(* Logix 5000 project; controller reports 1756-L63 rev 20.11; software revision 20.04; part 28 of 52 *)

        [2013].time.Year := 2023, [2013].time.Month := 1, [2013].time.Day := 16, [2013].time.Hour := 16, [2013].time.Minute := 9, [2013].time.Second := 59, [2014].log_data[0].min := 1.0, [2014].log_data[0].max := 1.0, [2014].log_data[0].total := 300.0, [2014].log_data[0].time := 300.0, [2014].log_data[0].minminute := 10, [2014].log_data[0].maxminute := 10, [2014].log_data[0].valid := 1, [2014].log_data[1].valid := 1, [2014].log_data[2].valid := 1, [2014].log_data[3].valid := 1, [2014].log_data[4].valid := 1, [2014].log_data[5].valid := 1, [2014].log_data[6].valid := 1, [2014].log_data[7].valid := 1, [2014].log_data[8].valid := 1, [2014].log_data[9].valid := 1, [2014].log_data[10].valid := 1, [2014].log_data[11].valid := 1, [2014].log_data[12].valid := 1, [2014].log_data[13].valid := 1, [2014].log_data[14].valid := 1, [2014].log_data[15].valid := 1, [2014].log_data[16].valid := 1, [2014].log_data[17].valid := 1, [2014].log_data[18].valid := 1, [2014].log_data[19].valid := 1, [2014].time.Year := 2023, [2014].time.Month := 1, [2014].time.Day := 16, [2014].time.Hour := 16, [2014].time.Minute := 14, [2014].time.Second := 59, [2015].log_data[0].min := 1.0, [2015].log_data[0].max := 1.0, [2015].log_data[0].total := 300.0, [2015].log_data[0].time := 300.0, [2015].log_data[0].minminute := 15, [2015].log_data[0].maxminute := 15, [2015].log_data[0].valid := 1, [2015].log_data[1].valid := 1, [2015].log_data[2].valid := 1, [2015].log_data[3].valid := 1, [2015].log_data[4].valid := 1, [2015].log_data[5].valid := 1, [2015].log_data[6].valid := 1, [2015].log_data[7].valid := 1, [2015].log_data[8].valid := 1, [2015].log_data[9].valid := 1, [2015].log_data[10].valid := 1, [2015].log_data[11].valid := 1, [2015].log_data[12].valid := 1, [2015].log_data[13].valid := 1, [2015].log_data[14].valid := 1, [2015].log_data[15].valid := 1,
        [2015].log_data[16].valid := 1, [2015].log_data[17].valid := 1, [2015].log_data[18].valid := 1, [2015].log_data[19].valid := 1, [2015].time.Year := 2023, [2015].time.Month := 1, [2015].time.Day := 16, [2015].time.Hour := 16, [2015].time.Minute := 19, [2015].time.Second := 59, [2016].log_data[0].min := 1.0, [2016].log_data[0].max := 1.0, [2016].log_data[0].total := 300.0, [2016].log_data[0].time := 300.0, [2016].log_data[0].minminute := 20, [2016].log_data[0].maxminute := 20, [2016].log_data[0].valid := 1, [2016].log_data[1].valid := 1, [2016].log_data[2].valid := 1, [2016].log_data[3].valid := 1, [2016].log_data[4].valid := 1, [2016].log_data[5].valid := 1, [2016].log_data[6].valid := 1, [2016].log_data[7].valid := 1, [2016].log_data[8].valid := 1, [2016].log_data[9].valid := 1, [2016].log_data[10].valid := 1, [2016].log_data[11].valid := 1, [2016].log_data[12].valid := 1, [2016].log_data[13].valid := 1, [2016].log_data[14].valid := 1, [2016].log_data[15].valid := 1, [2016].log_data[16].valid := 1, [2016].log_data[17].valid := 1, [2016].log_data[18].valid := 1, [2016].log_data[19].valid := 1, [2016].time.Year := 2023, [2016].time.Month := 1, [2016].time.Day := 16, [2016].time.Hour := 16, [2016].time.Minute := 24, [2016].time.Second := 59, [2017].log_data[0].min := 1.0, [2017].log_data[0].max := 1.0, [2017].log_data[0].total := 300.0, [2017].log_data[0].time := 300.0, [2017].log_data[0].minminute := 25, [2017].log_data[0].maxminute := 25, [2017].log_data[0].valid := 1, [2017].log_data[1].valid := 1, [2017].log_data[2].valid := 1, [2017].log_data[3].valid := 1, [2017].log_data[4].valid := 1, [2017].log_data[5].valid := 1, [2017].log_data[6].valid := 1, [2017].log_data[7].valid := 1, [2017].log_data[8].valid := 1, [2017].log_data[9].valid := 1, [2017].log_data[10].valid := 1, [2017].log_data[11].valid := 1,
        [2017].log_data[12].valid := 1, [2017].log_data[13].valid := 1, [2017].log_data[14].valid := 1, [2017].log_data[15].valid := 1, [2017].log_data[16].valid := 1, [2017].log_data[17].valid := 1, [2017].log_data[18].valid := 1, [2017].log_data[19].valid := 1, [2017].time.Year := 2023, [2017].time.Month := 1, [2017].time.Day := 16, [2017].time.Hour := 16, [2017].time.Minute := 29, [2017].time.Second := 59, [2018].log_data[0].min := 1.0, [2018].log_data[0].max := 1.0, [2018].log_data[0].total := 300.0, [2018].log_data[0].time := 300.0, [2018].log_data[0].minminute := 30, [2018].log_data[0].maxminute := 30, [2018].log_data[0].valid := 1, [2018].log_data[1].valid := 1, [2018].log_data[2].valid := 1, [2018].log_data[3].valid := 1, [2018].log_data[4].valid := 1, [2018].log_data[5].valid := 1, [2018].log_data[6].valid := 1, [2018].log_data[7].valid := 1, [2018].log_data[8].valid := 1, [2018].log_data[9].valid := 1, [2018].log_data[10].valid := 1, [2018].log_data[11].valid := 1, [2018].log_data[12].valid := 1, [2018].log_data[13].valid := 1, [2018].log_data[14].valid := 1, [2018].log_data[15].valid := 1, [2018].log_data[16].valid := 1, [2018].log_data[17].valid := 1, [2018].log_data[18].valid := 1, [2018].log_data[19].valid := 1, [2018].time.Year := 2023, [2018].time.Month := 1, [2018].time.Day := 16, [2018].time.Hour := 16, [2018].time.Minute := 34, [2018].time.Second := 59, [2019].log_data[0].min := 1.0, [2019].log_data[0].max := 1.0, [2019].log_data[0].total := 300.0, [2019].log_data[0].time := 300.0, [2019].log_data[0].minminute := 35, [2019].log_data[0].maxminute := 35, [2019].log_data[0].valid := 1, [2019].log_data[1].valid := 1, [2019].log_data[2].valid := 1, [2019].log_data[3].valid := 1, [2019].log_data[4].valid := 1, [2019].log_data[5].valid := 1, [2019].log_data[6].valid := 1, [2019].log_data[7].valid := 1,
        [2019].log_data[8].valid := 1, [2019].log_data[9].valid := 1, [2019].log_data[10].valid := 1, [2019].log_data[11].valid := 1, [2019].log_data[12].valid := 1, [2019].log_data[13].valid := 1, [2019].log_data[14].valid := 1, [2019].log_data[15].valid := 1, [2019].log_data[16].valid := 1, [2019].log_data[17].valid := 1, [2019].log_data[18].valid := 1, [2019].log_data[19].valid := 1, [2019].time.Year := 2023, [2019].time.Month := 1, [2019].time.Day := 16, [2019].time.Hour := 16, [2019].time.Minute := 39, [2019].time.Second := 59, [2020].log_data[0].min := 1.0, [2020].log_data[0].max := 1.0, [2020].log_data[0].total := 300.0, [2020].log_data[0].time := 300.0, [2020].log_data[0].minminute := 40, [2020].log_data[0].maxminute := 40, [2020].log_data[0].valid := 1, [2020].log_data[1].valid := 1, [2020].log_data[2].valid := 1, [2020].log_data[3].valid := 1, [2020].log_data[4].valid := 1, [2020].log_data[5].valid := 1, [2020].log_data[6].valid := 1, [2020].log_data[7].valid := 1, [2020].log_data[8].valid := 1, [2020].log_data[9].valid := 1, [2020].log_data[10].valid := 1, [2020].log_data[11].valid := 1, [2020].log_data[12].valid := 1, [2020].log_data[13].valid := 1, [2020].log_data[14].valid := 1, [2020].log_data[15].valid := 1, [2020].log_data[16].valid := 1, [2020].log_data[17].valid := 1, [2020].log_data[18].valid := 1, [2020].log_data[19].valid := 1, [2020].time.Year := 2023, [2020].time.Month := 1, [2020].time.Day := 16, [2020].time.Hour := 16, [2020].time.Minute := 44, [2020].time.Second := 59, [2021].log_data[0].min := 1.0, [2021].log_data[0].max := 1.0, [2021].log_data[0].total := 300.0, [2021].log_data[0].time := 300.0, [2021].log_data[0].minminute := 45, [2021].log_data[0].maxminute := 45, [2021].log_data[0].valid := 1, [2021].log_data[1].valid := 1, [2021].log_data[2].valid := 1, [2021].log_data[3].valid := 1,
        [2021].log_data[4].valid := 1, [2021].log_data[5].valid := 1, [2021].log_data[6].valid := 1, [2021].log_data[7].valid := 1, [2021].log_data[8].valid := 1, [2021].log_data[9].valid := 1, [2021].log_data[10].valid := 1, [2021].log_data[11].valid := 1, [2021].log_data[12].valid := 1, [2021].log_data[13].valid := 1, [2021].log_data[14].valid := 1, [2021].log_data[15].valid := 1, [2021].log_data[16].valid := 1, [2021].log_data[17].valid := 1, [2021].log_data[18].valid := 1, [2021].log_data[19].valid := 1, [2021].time.Year := 2023, [2021].time.Month := 1, [2021].time.Day := 16, [2021].time.Hour := 16, [2021].time.Minute := 49, [2021].time.Second := 59, [2022].log_data[0].min := 1.0, [2022].log_data[0].max := 1.0, [2022].log_data[0].total := 300.0, [2022].log_data[0].time := 300.0, [2022].log_data[0].minminute := 50, [2022].log_data[0].maxminute := 50, [2022].log_data[0].valid := 1, [2022].log_data[1].valid := 1, [2022].log_data[2].valid := 1, [2022].log_data[3].valid := 1, [2022].log_data[4].valid := 1, [2022].log_data[5].valid := 1, [2022].log_data[6].valid := 1, [2022].log_data[7].valid := 1, [2022].log_data[8].valid := 1, [2022].log_data[9].valid := 1, [2022].log_data[10].valid := 1, [2022].log_data[11].valid := 1, [2022].log_data[12].valid := 1, [2022].log_data[13].valid := 1, [2022].log_data[14].valid := 1, [2022].log_data[15].valid := 1, [2022].log_data[16].valid := 1, [2022].log_data[17].valid := 1, [2022].log_data[18].valid := 1, [2022].log_data[19].valid := 1, [2022].time.Year := 2023, [2022].time.Month := 1, [2022].time.Day := 16, [2022].time.Hour := 16, [2022].time.Minute := 54, [2022].time.Second := 59, [2023].log_data[0].min := 1.0, [2023].log_data[0].max := 1.0, [2023].log_data[0].total := 300.0, [2023].log_data[0].time := 300.0, [2023].log_data[0].minminute := 55, [2023].log_data[0].maxminute := 55,
        [2023].log_data[0].valid := 1, [2023].log_data[1].valid := 1, [2023].log_data[2].valid := 1, [2023].log_data[3].valid := 1, [2023].log_data[4].valid := 1, [2023].log_data[5].valid := 1, [2023].log_data[6].valid := 1, [2023].log_data[7].valid := 1, [2023].log_data[8].valid := 1, [2023].log_data[9].valid := 1, [2023].log_data[10].valid := 1, [2023].log_data[11].valid := 1, [2023].log_data[12].valid := 1, [2023].log_data[13].valid := 1, [2023].log_data[14].valid := 1, [2023].log_data[15].valid := 1, [2023].log_data[16].valid := 1, [2023].log_data[17].valid := 1, [2023].log_data[18].valid := 1, [2023].log_data[19].valid := 1, [2023].time.Year := 2023, [2023].time.Month := 1, [2023].time.Day := 16, [2023].time.Hour := 16, [2023].time.Minute := 59, [2023].time.Second := 59, [2024].log_data[0].min := 1.0, [2024].log_data[0].max := 1.0, [2024].log_data[0].total := 300.0, [2024].log_data[0].time := 300.0, [2024].log_data[0].valid := 1, [2024].log_data[1].valid := 1, [2024].log_data[2].valid := 1, [2024].log_data[3].valid := 1, [2024].log_data[4].valid := 1, [2024].log_data[5].valid := 1, [2024].log_data[6].valid := 1, [2024].log_data[7].valid := 1, [2024].log_data[8].valid := 1, [2024].log_data[9].valid := 1, [2024].log_data[10].valid := 1, [2024].log_data[11].valid := 1, [2024].log_data[12].valid := 1, [2024].log_data[13].valid := 1, [2024].log_data[14].valid := 1, [2024].log_data[15].valid := 1, [2024].log_data[16].valid := 1, [2024].log_data[17].valid := 1, [2024].log_data[18].valid := 1, [2024].log_data[19].valid := 1, [2024].time.Year := 2023, [2024].time.Month := 1, [2024].time.Day := 16, [2024].time.Hour := 17, [2024].time.Minute := 4, [2024].time.Second := 59, [2025].log_data[0].min := 1.0, [2025].log_data[0].max := 1.0, [2025].log_data[0].total := 300.0, [2025].log_data[0].time := 300.0,
        [2025].log_data[0].minminute := 5, [2025].log_data[0].maxminute := 5, [2025].log_data[0].valid := 1, [2025].log_data[1].valid := 1, [2025].log_data[2].valid := 1, [2025].log_data[3].valid := 1, [2025].log_data[4].valid := 1, [2025].log_data[5].valid := 1, [2025].log_data[6].valid := 1, [2025].log_data[7].valid := 1, [2025].log_data[8].valid := 1, [2025].log_data[9].valid := 1, [2025].log_data[10].valid := 1, [2025].log_data[11].valid := 1, [2025].log_data[12].valid := 1, [2025].log_data[13].valid := 1, [2025].log_data[14].valid := 1, [2025].log_data[15].valid := 1, [2025].log_data[16].valid := 1, [2025].log_data[17].valid := 1, [2025].log_data[18].valid := 1, [2025].log_data[19].valid := 1, [2025].time.Year := 2023, [2025].time.Month := 1, [2025].time.Day := 16, [2025].time.Hour := 17, [2025].time.Minute := 9, [2025].time.Second := 59, [2026].log_data[0].min := 1.0, [2026].log_data[0].max := 1.0, [2026].log_data[0].total := 300.0, [2026].log_data[0].time := 300.0, [2026].log_data[0].minminute := 10, [2026].log_data[0].maxminute := 10, [2026].log_data[0].valid := 1, [2026].log_data[1].valid := 1, [2026].log_data[2].valid := 1, [2026].log_data[3].valid := 1, [2026].log_data[4].valid := 1, [2026].log_data[5].valid := 1, [2026].log_data[6].valid := 1, [2026].log_data[7].valid := 1, [2026].log_data[8].valid := 1, [2026].log_data[9].valid := 1, [2026].log_data[10].valid := 1, [2026].log_data[11].valid := 1, [2026].log_data[12].valid := 1, [2026].log_data[13].valid := 1, [2026].log_data[14].valid := 1, [2026].log_data[15].valid := 1, [2026].log_data[16].valid := 1, [2026].log_data[17].valid := 1, [2026].log_data[18].valid := 1, [2026].log_data[19].valid := 1, [2026].time.Year := 2023, [2026].time.Month := 1, [2026].time.Day := 16, [2026].time.Hour := 17, [2026].time.Minute := 14, [2026].time.Second := 59,
        [2027].log_data[0].min := 1.0, [2027].log_data[0].max := 1.0, [2027].log_data[0].total := 300.0, [2027].log_data[0].time := 300.0, [2027].log_data[0].minminute := 15, [2027].log_data[0].maxminute := 15, [2027].log_data[0].valid := 1, [2027].log_data[1].valid := 1, [2027].log_data[2].valid := 1, [2027].log_data[3].valid := 1, [2027].log_data[4].valid := 1, [2027].log_data[5].valid := 1, [2027].log_data[6].valid := 1, [2027].log_data[7].valid := 1, [2027].log_data[8].valid := 1, [2027].log_data[9].valid := 1, [2027].log_data[10].valid := 1, [2027].log_data[11].valid := 1, [2027].log_data[12].valid := 1, [2027].log_data[13].valid := 1, [2027].log_data[14].valid := 1, [2027].log_data[15].valid := 1, [2027].log_data[16].valid := 1, [2027].log_data[17].valid := 1, [2027].log_data[18].valid := 1, [2027].log_data[19].valid := 1, [2027].time.Year := 2023, [2027].time.Month := 1, [2027].time.Day := 16, [2027].time.Hour := 17, [2027].time.Minute := 19, [2027].time.Second := 59, [2028].log_data[0].min := 1.0, [2028].log_data[0].max := 1.0, [2028].log_data[0].total := 300.0, [2028].log_data[0].time := 300.0, [2028].log_data[0].minminute := 20, [2028].log_data[0].maxminute := 20, [2028].log_data[0].valid := 1, [2028].log_data[1].valid := 1, [2028].log_data[2].valid := 1, [2028].log_data[3].valid := 1, [2028].log_data[4].valid := 1, [2028].log_data[5].valid := 1, [2028].log_data[6].valid := 1, [2028].log_data[7].valid := 1, [2028].log_data[8].valid := 1, [2028].log_data[9].valid := 1, [2028].log_data[10].valid := 1, [2028].log_data[11].valid := 1, [2028].log_data[12].valid := 1, [2028].log_data[13].valid := 1, [2028].log_data[14].valid := 1, [2028].log_data[15].valid := 1, [2028].log_data[16].valid := 1, [2028].log_data[17].valid := 1, [2028].log_data[18].valid := 1, [2028].log_data[19].valid := 1, [2028].time.Year := 2023, [2028].time.Month := 1,
        [2028].time.Day := 16, [2028].time.Hour := 17, [2028].time.Minute := 24, [2028].time.Second := 59, [2029].log_data[0].min := 1.0, [2029].log_data[0].max := 1.0, [2029].log_data[0].total := 300.0, [2029].log_data[0].time := 300.0, [2029].log_data[0].minminute := 25, [2029].log_data[0].maxminute := 25, [2029].log_data[0].valid := 1, [2029].log_data[1].valid := 1, [2029].log_data[2].valid := 1, [2029].log_data[3].valid := 1, [2029].log_data[4].valid := 1, [2029].log_data[5].valid := 1, [2029].log_data[6].valid := 1, [2029].log_data[7].valid := 1, [2029].log_data[8].valid := 1, [2029].log_data[9].valid := 1, [2029].log_data[10].valid := 1, [2029].log_data[11].valid := 1, [2029].log_data[12].valid := 1, [2029].log_data[13].valid := 1, [2029].log_data[14].valid := 1, [2029].log_data[15].valid := 1, [2029].log_data[16].valid := 1, [2029].log_data[17].valid := 1, [2029].log_data[18].valid := 1, [2029].log_data[19].valid := 1, [2029].time.Year := 2023, [2029].time.Month := 1, [2029].time.Day := 16, [2029].time.Hour := 17, [2029].time.Minute := 29, [2029].time.Second := 59, [2030].log_data[0].min := 1.0, [2030].log_data[0].max := 1.0, [2030].log_data[0].total := 300.0, [2030].log_data[0].time := 300.0, [2030].log_data[0].minminute := 30, [2030].log_data[0].maxminute := 30, [2030].log_data[0].valid := 1, [2030].log_data[1].valid := 1, [2030].log_data[2].valid := 1, [2030].log_data[3].valid := 1, [2030].log_data[4].valid := 1, [2030].log_data[5].valid := 1, [2030].log_data[6].valid := 1, [2030].log_data[7].valid := 1, [2030].log_data[8].valid := 1, [2030].log_data[9].valid := 1, [2030].log_data[10].valid := 1, [2030].log_data[11].valid := 1, [2030].log_data[12].valid := 1, [2030].log_data[13].valid := 1, [2030].log_data[14].valid := 1, [2030].log_data[15].valid := 1, [2030].log_data[16].valid := 1, [2030].log_data[17].valid := 1,
        [2030].log_data[18].valid := 1, [2030].log_data[19].valid := 1, [2030].time.Year := 2023, [2030].time.Month := 1, [2030].time.Day := 16, [2030].time.Hour := 17, [2030].time.Minute := 34, [2030].time.Second := 59, [2031].log_data[0].min := 1.0, [2031].log_data[0].max := 1.0, [2031].log_data[0].total := 300.0, [2031].log_data[0].time := 300.0, [2031].log_data[0].minminute := 35, [2031].log_data[0].maxminute := 35, [2031].log_data[0].valid := 1, [2031].log_data[1].valid := 1, [2031].log_data[2].valid := 1, [2031].log_data[3].valid := 1, [2031].log_data[4].valid := 1, [2031].log_data[5].valid := 1, [2031].log_data[6].valid := 1, [2031].log_data[7].valid := 1, [2031].log_data[8].valid := 1, [2031].log_data[9].valid := 1, [2031].log_data[10].valid := 1, [2031].log_data[11].valid := 1, [2031].log_data[12].valid := 1, [2031].log_data[13].valid := 1, [2031].log_data[14].valid := 1, [2031].log_data[15].valid := 1, [2031].log_data[16].valid := 1, [2031].log_data[17].valid := 1, [2031].log_data[18].valid := 1, [2031].log_data[19].valid := 1, [2031].time.Year := 2023, [2031].time.Month := 1, [2031].time.Day := 16, [2031].time.Hour := 17, [2031].time.Minute := 39, [2031].time.Second := 59, [2032].log_data[0].min := 1.0, [2032].log_data[0].max := 1.0, [2032].log_data[0].total := 300.0, [2032].log_data[0].time := 300.0, [2032].log_data[0].minminute := 40, [2032].log_data[0].maxminute := 40, [2032].log_data[0].valid := 1, [2032].log_data[1].valid := 1, [2032].log_data[2].valid := 1, [2032].log_data[3].valid := 1, [2032].log_data[4].valid := 1, [2032].log_data[5].valid := 1, [2032].log_data[6].valid := 1, [2032].log_data[7].valid := 1, [2032].log_data[8].valid := 1, [2032].log_data[9].valid := 1, [2032].log_data[10].valid := 1, [2032].log_data[11].valid := 1, [2032].log_data[12].valid := 1, [2032].log_data[13].valid := 1,
        [2032].log_data[14].valid := 1, [2032].log_data[15].valid := 1, [2032].log_data[16].valid := 1, [2032].log_data[17].valid := 1, [2032].log_data[18].valid := 1, [2032].log_data[19].valid := 1, [2032].time.Year := 2023, [2032].time.Month := 1, [2032].time.Day := 16, [2032].time.Hour := 17, [2032].time.Minute := 44, [2032].time.Second := 59, [2033].log_data[0].min := 1.0, [2033].log_data[0].max := 1.0, [2033].log_data[0].total := 300.0, [2033].log_data[0].time := 300.0, [2033].log_data[0].minminute := 45, [2033].log_data[0].maxminute := 45, [2033].log_data[0].valid := 1, [2033].log_data[1].valid := 1, [2033].log_data[2].valid := 1, [2033].log_data[3].valid := 1, [2033].log_data[4].valid := 1, [2033].log_data[5].valid := 1, [2033].log_data[6].valid := 1, [2033].log_data[7].valid := 1, [2033].log_data[8].valid := 1, [2033].log_data[9].valid := 1, [2033].log_data[10].valid := 1, [2033].log_data[11].valid := 1, [2033].log_data[12].valid := 1, [2033].log_data[13].valid := 1, [2033].log_data[14].valid := 1, [2033].log_data[15].valid := 1, [2033].log_data[16].valid := 1, [2033].log_data[17].valid := 1, [2033].log_data[18].valid := 1, [2033].log_data[19].valid := 1, [2033].time.Year := 2023, [2033].time.Month := 1, [2033].time.Day := 16, [2033].time.Hour := 17, [2033].time.Minute := 49, [2033].time.Second := 59, [2034].log_data[0].min := 1.0, [2034].log_data[0].max := 1.0, [2034].log_data[0].total := 300.0, [2034].log_data[0].time := 300.0, [2034].log_data[0].minminute := 50, [2034].log_data[0].maxminute := 50, [2034].log_data[0].valid := 1, [2034].log_data[1].valid := 1, [2034].log_data[2].valid := 1, [2034].log_data[3].valid := 1, [2034].log_data[4].valid := 1, [2034].log_data[5].valid := 1, [2034].log_data[6].valid := 1, [2034].log_data[7].valid := 1, [2034].log_data[8].valid := 1, [2034].log_data[9].valid := 1,
        [2034].log_data[10].valid := 1, [2034].log_data[11].valid := 1, [2034].log_data[12].valid := 1, [2034].log_data[13].valid := 1, [2034].log_data[14].valid := 1, [2034].log_data[15].valid := 1, [2034].log_data[16].valid := 1, [2034].log_data[17].valid := 1, [2034].log_data[18].valid := 1, [2034].log_data[19].valid := 1, [2034].time.Year := 2023, [2034].time.Month := 1, [2034].time.Day := 16, [2034].time.Hour := 17, [2034].time.Minute := 54, [2034].time.Second := 59, [2035].log_data[0].min := 1.0, [2035].log_data[0].max := 1.0, [2035].log_data[0].total := 300.0, [2035].log_data[0].time := 300.0, [2035].log_data[0].minminute := 55, [2035].log_data[0].maxminute := 55, [2035].log_data[0].valid := 1, [2035].log_data[1].valid := 1, [2035].log_data[2].valid := 1, [2035].log_data[3].valid := 1, [2035].log_data[4].valid := 1, [2035].log_data[5].valid := 1, [2035].log_data[6].valid := 1, [2035].log_data[7].valid := 1, [2035].log_data[8].valid := 1, [2035].log_data[9].valid := 1, [2035].log_data[10].valid := 1, [2035].log_data[11].valid := 1, [2035].log_data[12].valid := 1, [2035].log_data[13].valid := 1, [2035].log_data[14].valid := 1, [2035].log_data[15].valid := 1, [2035].log_data[16].valid := 1, [2035].log_data[17].valid := 1, [2035].log_data[18].valid := 1, [2035].log_data[19].valid := 1, [2035].time.Year := 2023, [2035].time.Month := 1, [2035].time.Day := 16, [2035].time.Hour := 17, [2035].time.Minute := 59, [2035].time.Second := 59, [2036].log_data[0].min := 1.0, [2036].log_data[0].max := 1.0, [2036].log_data[0].total := 300.0, [2036].log_data[0].time := 300.0, [2036].log_data[0].valid := 1, [2036].log_data[1].valid := 1, [2036].log_data[2].valid := 1, [2036].log_data[3].valid := 1, [2036].log_data[4].valid := 1, [2036].log_data[5].valid := 1, [2036].log_data[6].valid := 1, [2036].log_data[7].valid := 1,
        [2036].log_data[8].valid := 1, [2036].log_data[9].valid := 1, [2036].log_data[10].valid := 1, [2036].log_data[11].valid := 1, [2036].log_data[12].valid := 1, [2036].log_data[13].valid := 1, [2036].log_data[14].valid := 1, [2036].log_data[15].valid := 1, [2036].log_data[16].valid := 1, [2036].log_data[17].valid := 1, [2036].log_data[18].valid := 1, [2036].log_data[19].valid := 1, [2036].time.Year := 2023, [2036].time.Month := 1, [2036].time.Day := 16, [2036].time.Hour := 18, [2036].time.Minute := 4, [2036].time.Second := 59, [2037].log_data[0].min := 1.0, [2037].log_data[0].max := 1.0, [2037].log_data[0].total := 300.0, [2037].log_data[0].time := 300.0, [2037].log_data[0].minminute := 5, [2037].log_data[0].maxminute := 5, [2037].log_data[0].valid := 1, [2037].log_data[1].valid := 1, [2037].log_data[2].valid := 1, [2037].log_data[3].valid := 1, [2037].log_data[4].valid := 1, [2037].log_data[5].valid := 1, [2037].log_data[6].valid := 1, [2037].log_data[7].valid := 1, [2037].log_data[8].valid := 1, [2037].log_data[9].valid := 1, [2037].log_data[10].valid := 1, [2037].log_data[11].valid := 1, [2037].log_data[12].valid := 1, [2037].log_data[13].valid := 1, [2037].log_data[14].valid := 1, [2037].log_data[15].valid := 1, [2037].log_data[16].valid := 1, [2037].log_data[17].valid := 1, [2037].log_data[18].valid := 1, [2037].log_data[19].valid := 1, [2037].time.Year := 2023, [2037].time.Month := 1, [2037].time.Day := 16, [2037].time.Hour := 18, [2037].time.Minute := 9, [2037].time.Second := 59, [2038].log_data[0].min := 1.0, [2038].log_data[0].max := 1.0, [2038].log_data[0].total := 300.0, [2038].log_data[0].time := 300.0, [2038].log_data[0].minminute := 10, [2038].log_data[0].maxminute := 10, [2038].log_data[0].valid := 1, [2038].log_data[1].valid := 1, [2038].log_data[2].valid := 1, [2038].log_data[3].valid := 1,
        [2038].log_data[4].valid := 1, [2038].log_data[5].valid := 1, [2038].log_data[6].valid := 1, [2038].log_data[7].valid := 1, [2038].log_data[8].valid := 1, [2038].log_data[9].valid := 1, [2038].log_data[10].valid := 1, [2038].log_data[11].valid := 1, [2038].log_data[12].valid := 1, [2038].log_data[13].valid := 1, [2038].log_data[14].valid := 1, [2038].log_data[15].valid := 1, [2038].log_data[16].valid := 1, [2038].log_data[17].valid := 1, [2038].log_data[18].valid := 1, [2038].log_data[19].valid := 1, [2038].time.Year := 2023, [2038].time.Month := 1, [2038].time.Day := 16, [2038].time.Hour := 18, [2038].time.Minute := 14, [2038].time.Second := 59, [2039].log_data[0].min := 1.0, [2039].log_data[0].max := 1.0, [2039].log_data[0].total := 300.0, [2039].log_data[0].time := 300.0, [2039].log_data[0].minminute := 15, [2039].log_data[0].maxminute := 15, [2039].log_data[0].valid := 1, [2039].log_data[1].valid := 1, [2039].log_data[2].valid := 1, [2039].log_data[3].valid := 1, [2039].log_data[4].valid := 1, [2039].log_data[5].valid := 1, [2039].log_data[6].valid := 1, [2039].log_data[7].valid := 1, [2039].log_data[8].valid := 1, [2039].log_data[9].valid := 1, [2039].log_data[10].valid := 1, [2039].log_data[11].valid := 1, [2039].log_data[12].valid := 1, [2039].log_data[13].valid := 1, [2039].log_data[14].valid := 1, [2039].log_data[15].valid := 1, [2039].log_data[16].valid := 1, [2039].log_data[17].valid := 1, [2039].log_data[18].valid := 1, [2039].log_data[19].valid := 1, [2039].time.Year := 2023, [2039].time.Month := 1, [2039].time.Day := 16, [2039].time.Hour := 18, [2039].time.Minute := 19, [2039].time.Second := 59, [2040].log_data[0].min := 1.0, [2040].log_data[0].max := 1.0, [2040].log_data[0].total := 300.0, [2040].log_data[0].time := 300.0, [2040].log_data[0].minminute := 20, [2040].log_data[0].maxminute := 20,
        [2040].log_data[0].valid := 1, [2040].log_data[1].valid := 1, [2040].log_data[2].valid := 1, [2040].log_data[3].valid := 1, [2040].log_data[4].valid := 1, [2040].log_data[5].valid := 1, [2040].log_data[6].valid := 1, [2040].log_data[7].valid := 1, [2040].log_data[8].valid := 1, [2040].log_data[9].valid := 1, [2040].log_data[10].valid := 1, [2040].log_data[11].valid := 1, [2040].log_data[12].valid := 1, [2040].log_data[13].valid := 1, [2040].log_data[14].valid := 1, [2040].log_data[15].valid := 1, [2040].log_data[16].valid := 1, [2040].log_data[17].valid := 1, [2040].log_data[18].valid := 1, [2040].log_data[19].valid := 1, [2040].time.Year := 2023, [2040].time.Month := 1, [2040].time.Day := 16, [2040].time.Hour := 18, [2040].time.Minute := 24, [2040].time.Second := 59, [2041].log_data[0].min := 1.0, [2041].log_data[0].max := 1.0, [2041].log_data[0].total := 300.0, [2041].log_data[0].time := 300.0, [2041].log_data[0].minminute := 25, [2041].log_data[0].maxminute := 25, [2041].log_data[0].valid := 1, [2041].log_data[1].valid := 1, [2041].log_data[2].valid := 1, [2041].log_data[3].valid := 1, [2041].log_data[4].valid := 1, [2041].log_data[5].valid := 1, [2041].log_data[6].valid := 1, [2041].log_data[7].valid := 1, [2041].log_data[8].valid := 1, [2041].log_data[9].valid := 1, [2041].log_data[10].valid := 1, [2041].log_data[11].valid := 1, [2041].log_data[12].valid := 1, [2041].log_data[13].valid := 1, [2041].log_data[14].valid := 1, [2041].log_data[15].valid := 1, [2041].log_data[16].valid := 1, [2041].log_data[17].valid := 1, [2041].log_data[18].valid := 1, [2041].log_data[19].valid := 1, [2041].time.Year := 2023, [2041].time.Month := 1, [2041].time.Day := 16, [2041].time.Hour := 18, [2041].time.Minute := 29, [2041].time.Second := 59, [2042].log_data[0].min := 1.0, [2042].log_data[0].max := 1.0,
        [2042].log_data[0].total := 300.0, [2042].log_data[0].time := 300.0, [2042].log_data[0].minminute := 30, [2042].log_data[0].maxminute := 30, [2042].log_data[0].valid := 1, [2042].log_data[1].valid := 1, [2042].log_data[2].valid := 1, [2042].log_data[3].valid := 1, [2042].log_data[4].valid := 1, [2042].log_data[5].valid := 1, [2042].log_data[6].valid := 1, [2042].log_data[7].valid := 1, [2042].log_data[8].valid := 1, [2042].log_data[9].valid := 1, [2042].log_data[10].valid := 1, [2042].log_data[11].valid := 1, [2042].log_data[12].valid := 1, [2042].log_data[13].valid := 1, [2042].log_data[14].valid := 1, [2042].log_data[15].valid := 1, [2042].log_data[16].valid := 1, [2042].log_data[17].valid := 1, [2042].log_data[18].valid := 1, [2042].log_data[19].valid := 1, [2042].time.Year := 2023, [2042].time.Month := 1, [2042].time.Day := 16, [2042].time.Hour := 18, [2042].time.Minute := 34, [2042].time.Second := 59, [2043].log_data[0].min := 1.0, [2043].log_data[0].max := 1.0, [2043].log_data[0].total := 300.0, [2043].log_data[0].time := 300.0, [2043].log_data[0].minminute := 35, [2043].log_data[0].maxminute := 35, [2043].log_data[0].valid := 1, [2043].log_data[1].valid := 1, [2043].log_data[2].valid := 1, [2043].log_data[3].valid := 1, [2043].log_data[4].valid := 1, [2043].log_data[5].valid := 1, [2043].log_data[6].valid := 1, [2043].log_data[7].valid := 1, [2043].log_data[8].valid := 1, [2043].log_data[9].valid := 1, [2043].log_data[10].valid := 1, [2043].log_data[11].valid := 1, [2043].log_data[12].valid := 1, [2043].log_data[13].valid := 1, [2043].log_data[14].valid := 1, [2043].log_data[15].valid := 1, [2043].log_data[16].valid := 1, [2043].log_data[17].valid := 1, [2043].log_data[18].valid := 1, [2043].log_data[19].valid := 1, [2043].time.Year := 2023, [2043].time.Month := 1, [2043].time.Day := 16, [2043].time.Hour := 18,
        [2043].time.Minute := 39, [2043].time.Second := 59, [2044].log_data[0].min := 1.0, [2044].log_data[0].max := 1.0, [2044].log_data[0].total := 300.0, [2044].log_data[0].time := 300.0, [2044].log_data[0].minminute := 40, [2044].log_data[0].maxminute := 40, [2044].log_data[0].valid := 1, [2044].log_data[1].valid := 1, [2044].log_data[2].valid := 1, [2044].log_data[3].valid := 1, [2044].log_data[4].valid := 1, [2044].log_data[5].valid := 1, [2044].log_data[6].valid := 1, [2044].log_data[7].valid := 1, [2044].log_data[8].valid := 1, [2044].log_data[9].valid := 1, [2044].log_data[10].valid := 1, [2044].log_data[11].valid := 1, [2044].log_data[12].valid := 1, [2044].log_data[13].valid := 1, [2044].log_data[14].valid := 1, [2044].log_data[15].valid := 1, [2044].log_data[16].valid := 1, [2044].log_data[17].valid := 1, [2044].log_data[18].valid := 1, [2044].log_data[19].valid := 1, [2044].time.Year := 2023, [2044].time.Month := 1, [2044].time.Day := 16, [2044].time.Hour := 18, [2044].time.Minute := 44, [2044].time.Second := 59, [2045].log_data[0].min := 1.0, [2045].log_data[0].max := 1.0, [2045].log_data[0].total := 300.0, [2045].log_data[0].time := 300.0, [2045].log_data[0].minminute := 45, [2045].log_data[0].maxminute := 45, [2045].log_data[0].valid := 1, [2045].log_data[1].valid := 1, [2045].log_data[2].valid := 1, [2045].log_data[3].valid := 1, [2045].log_data[4].valid := 1, [2045].log_data[5].valid := 1, [2045].log_data[6].valid := 1, [2045].log_data[7].valid := 1, [2045].log_data[8].valid := 1, [2045].log_data[9].valid := 1, [2045].log_data[10].valid := 1, [2045].log_data[11].valid := 1, [2045].log_data[12].valid := 1, [2045].log_data[13].valid := 1, [2045].log_data[14].valid := 1, [2045].log_data[15].valid := 1, [2045].log_data[16].valid := 1, [2045].log_data[17].valid := 1, [2045].log_data[18].valid := 1, [2045].log_data[19].valid := 1,
        [2045].time.Year := 2023, [2045].time.Month := 1, [2045].time.Day := 16, [2045].time.Hour := 18, [2045].time.Minute := 49, [2045].time.Second := 59, [2046].log_data[0].min := 1.0, [2046].log_data[0].max := 1.0, [2046].log_data[0].total := 300.0, [2046].log_data[0].time := 300.0, [2046].log_data[0].minminute := 50, [2046].log_data[0].maxminute := 50, [2046].log_data[0].valid := 1, [2046].log_data[1].valid := 1, [2046].log_data[2].valid := 1, [2046].log_data[3].valid := 1, [2046].log_data[4].valid := 1, [2046].log_data[5].valid := 1, [2046].log_data[6].valid := 1, [2046].log_data[7].valid := 1, [2046].log_data[8].valid := 1, [2046].log_data[9].valid := 1, [2046].log_data[10].valid := 1, [2046].log_data[11].valid := 1, [2046].log_data[12].valid := 1, [2046].log_data[13].valid := 1, [2046].log_data[14].valid := 1, [2046].log_data[15].valid := 1, [2046].log_data[16].valid := 1, [2046].log_data[17].valid := 1, [2046].log_data[18].valid := 1, [2046].log_data[19].valid := 1, [2046].time.Year := 2023, [2046].time.Month := 1, [2046].time.Day := 16, [2046].time.Hour := 18, [2046].time.Minute := 54, [2046].time.Second := 59, [2047].log_data[0].min := 1.0, [2047].log_data[0].max := 1.0, [2047].log_data[0].total := 300.0, [2047].log_data[0].time := 300.0, [2047].log_data[0].minminute := 55, [2047].log_data[0].maxminute := 55, [2047].log_data[0].valid := 1, [2047].log_data[1].valid := 1, [2047].log_data[2].valid := 1, [2047].log_data[3].valid := 1, [2047].log_data[4].valid := 1, [2047].log_data[5].valid := 1, [2047].log_data[6].valid := 1, [2047].log_data[7].valid := 1, [2047].log_data[8].valid := 1, [2047].log_data[9].valid := 1, [2047].log_data[10].valid := 1, [2047].log_data[11].valid := 1, [2047].log_data[12].valid := 1, [2047].log_data[13].valid := 1, [2047].log_data[14].valid := 1, [2047].log_data[15].valid := 1,
        [2047].log_data[16].valid := 1, [2047].log_data[17].valid := 1, [2047].log_data[18].valid := 1, [2047].log_data[19].valid := 1, [2047].time.Year := 2023, [2047].time.Month := 1, [2047].time.Day := 16, [2047].time.Hour := 18, [2047].time.Minute := 59, [2047].time.Second := 59, [2048].log_data[0].min := 1.0, [2048].log_data[0].max := 1.0, [2048].log_data[0].total := 300.0, [2048].log_data[0].time := 300.0, [2048].log_data[0].valid := 1, [2048].log_data[1].valid := 1, [2048].log_data[2].valid := 1, [2048].log_data[3].valid := 1, [2048].log_data[4].valid := 1, [2048].log_data[5].valid := 1, [2048].log_data[6].valid := 1, [2048].log_data[7].valid := 1, [2048].log_data[8].valid := 1, [2048].log_data[9].valid := 1, [2048].log_data[10].valid := 1, [2048].log_data[11].valid := 1, [2048].log_data[12].valid := 1, [2048].log_data[13].valid := 1, [2048].log_data[14].valid := 1, [2048].log_data[15].valid := 1, [2048].log_data[16].valid := 1, [2048].log_data[17].valid := 1, [2048].log_data[18].valid := 1, [2048].log_data[19].valid := 1, [2048].time.Year := 2023, [2048].time.Month := 1, [2048].time.Day := 16, [2048].time.Hour := 19, [2048].time.Minute := 4, [2048].time.Second := 59, [2049].log_data[0].min := 1.0, [2049].log_data[0].max := 1.0, [2049].log_data[0].total := 300.0, [2049].log_data[0].time := 300.0, [2049].log_data[0].minminute := 5, [2049].log_data[0].maxminute := 5, [2049].log_data[0].valid := 1, [2049].log_data[1].valid := 1, [2049].log_data[2].valid := 1, [2049].log_data[3].valid := 1, [2049].log_data[4].valid := 1, [2049].log_data[5].valid := 1, [2049].log_data[6].valid := 1, [2049].log_data[7].valid := 1, [2049].log_data[8].valid := 1, [2049].log_data[9].valid := 1, [2049].log_data[10].valid := 1, [2049].log_data[11].valid := 1, [2049].log_data[12].valid := 1, [2049].log_data[13].valid := 1,
        [2049].log_data[14].valid := 1, [2049].log_data[15].valid := 1, [2049].log_data[16].valid := 1, [2049].log_data[17].valid := 1, [2049].log_data[18].valid := 1, [2049].log_data[19].valid := 1, [2049].time.Year := 2023, [2049].time.Month := 1, [2049].time.Day := 16, [2049].time.Hour := 19, [2049].time.Minute := 9, [2049].time.Second := 59, [2050].log_data[0].min := 1.0, [2050].log_data[0].max := 1.0, [2050].log_data[0].total := 300.0, [2050].log_data[0].time := 300.0, [2050].log_data[0].minminute := 10, [2050].log_data[0].maxminute := 10, [2050].log_data[0].valid := 1, [2050].log_data[1].valid := 1, [2050].log_data[2].valid := 1, [2050].log_data[3].valid := 1, [2050].log_data[4].valid := 1, [2050].log_data[5].valid := 1, [2050].log_data[6].valid := 1, [2050].log_data[7].valid := 1, [2050].log_data[8].valid := 1, [2050].log_data[9].valid := 1, [2050].log_data[10].valid := 1, [2050].log_data[11].valid := 1, [2050].log_data[12].valid := 1, [2050].log_data[13].valid := 1, [2050].log_data[14].valid := 1, [2050].log_data[15].valid := 1, [2050].log_data[16].valid := 1, [2050].log_data[17].valid := 1, [2050].log_data[18].valid := 1, [2050].log_data[19].valid := 1, [2050].time.Year := 2023, [2050].time.Month := 1, [2050].time.Day := 16, [2050].time.Hour := 19, [2050].time.Minute := 14, [2050].time.Second := 59, [2051].log_data[0].min := 1.0, [2051].log_data[0].max := 1.0, [2051].log_data[0].total := 300.0, [2051].log_data[0].time := 300.0, [2051].log_data[0].minminute := 15, [2051].log_data[0].maxminute := 15, [2051].log_data[0].valid := 1, [2051].log_data[1].valid := 1, [2051].log_data[2].valid := 1, [2051].log_data[3].valid := 1, [2051].log_data[4].valid := 1, [2051].log_data[5].valid := 1, [2051].log_data[6].valid := 1, [2051].log_data[7].valid := 1, [2051].log_data[8].valid := 1, [2051].log_data[9].valid := 1,
        [2051].log_data[10].valid := 1, [2051].log_data[11].valid := 1, [2051].log_data[12].valid := 1, [2051].log_data[13].valid := 1, [2051].log_data[14].valid := 1, [2051].log_data[15].valid := 1, [2051].log_data[16].valid := 1, [2051].log_data[17].valid := 1, [2051].log_data[18].valid := 1, [2051].log_data[19].valid := 1, [2051].time.Year := 2023, [2051].time.Month := 1, [2051].time.Day := 16, [2051].time.Hour := 19, [2051].time.Minute := 19, [2051].time.Second := 59, [2052].log_data[0].min := 1.0, [2052].log_data[0].max := 1.0, [2052].log_data[0].total := 300.0, [2052].log_data[0].time := 300.0, [2052].log_data[0].minminute := 20, [2052].log_data[0].maxminute := 20, [2052].log_data[0].valid := 1, [2052].log_data[1].valid := 1, [2052].log_data[2].valid := 1, [2052].log_data[3].valid := 1, [2052].log_data[4].valid := 1, [2052].log_data[5].valid := 1, [2052].log_data[6].valid := 1, [2052].log_data[7].valid := 1, [2052].log_data[8].valid := 1, [2052].log_data[9].valid := 1, [2052].log_data[10].valid := 1, [2052].log_data[11].valid := 1, [2052].log_data[12].valid := 1, [2052].log_data[13].valid := 1, [2052].log_data[14].valid := 1, [2052].log_data[15].valid := 1, [2052].log_data[16].valid := 1, [2052].log_data[17].valid := 1, [2052].log_data[18].valid := 1, [2052].log_data[19].valid := 1, [2052].time.Year := 2023, [2052].time.Month := 1, [2052].time.Day := 16, [2052].time.Hour := 19, [2052].time.Minute := 24, [2052].time.Second := 59, [2053].log_data[0].min := 1.0, [2053].log_data[0].max := 1.0, [2053].log_data[0].total := 300.0, [2053].log_data[0].time := 300.0, [2053].log_data[0].minminute := 25, [2053].log_data[0].maxminute := 25, [2053].log_data[0].valid := 1, [2053].log_data[1].valid := 1, [2053].log_data[2].valid := 1, [2053].log_data[3].valid := 1, [2053].log_data[4].valid := 1, [2053].log_data[5].valid := 1,
        [2053].log_data[6].valid := 1, [2053].log_data[7].valid := 1, [2053].log_data[8].valid := 1, [2053].log_data[9].valid := 1, [2053].log_data[10].valid := 1, [2053].log_data[11].valid := 1, [2053].log_data[12].valid := 1, [2053].log_data[13].valid := 1, [2053].log_data[14].valid := 1, [2053].log_data[15].valid := 1, [2053].log_data[16].valid := 1, [2053].log_data[17].valid := 1, [2053].log_data[18].valid := 1, [2053].log_data[19].valid := 1, [2053].time.Year := 2023, [2053].time.Month := 1, [2053].time.Day := 16, [2053].time.Hour := 19, [2053].time.Minute := 29, [2053].time.Second := 59, [2054].log_data[0].min := 1.0, [2054].log_data[0].max := 1.0, [2054].log_data[0].total := 300.0, [2054].log_data[0].time := 300.0, [2054].log_data[0].minminute := 30, [2054].log_data[0].maxminute := 30, [2054].log_data[0].valid := 1, [2054].log_data[1].valid := 1, [2054].log_data[2].valid := 1, [2054].log_data[3].valid := 1, [2054].log_data[4].valid := 1, [2054].log_data[5].valid := 1, [2054].log_data[6].valid := 1, [2054].log_data[7].valid := 1, [2054].log_data[8].valid := 1, [2054].log_data[9].valid := 1, [2054].log_data[10].valid := 1, [2054].log_data[11].valid := 1, [2054].log_data[12].valid := 1, [2054].log_data[13].valid := 1, [2054].log_data[14].valid := 1, [2054].log_data[15].valid := 1, [2054].log_data[16].valid := 1, [2054].log_data[17].valid := 1, [2054].log_data[18].valid := 1, [2054].log_data[19].valid := 1, [2054].time.Year := 2023, [2054].time.Month := 1, [2054].time.Day := 16, [2054].time.Hour := 19, [2054].time.Minute := 34, [2054].time.Second := 59, [2055].log_data[0].min := 1.0, [2055].log_data[0].max := 1.0, [2055].log_data[0].total := 300.0, [2055].log_data[0].time := 300.0, [2055].log_data[0].minminute := 35, [2055].log_data[0].maxminute := 35, [2055].log_data[0].valid := 1, [2055].log_data[1].valid := 1,
        [2055].log_data[2].valid := 1, [2055].log_data[3].valid := 1, [2055].log_data[4].valid := 1, [2055].log_data[5].valid := 1, [2055].log_data[6].valid := 1, [2055].log_data[7].valid := 1, [2055].log_data[8].valid := 1, [2055].log_data[9].valid := 1, [2055].log_data[10].valid := 1, [2055].log_data[11].valid := 1, [2055].log_data[12].valid := 1, [2055].log_data[13].valid := 1, [2055].log_data[14].valid := 1, [2055].log_data[15].valid := 1, [2055].log_data[16].valid := 1, [2055].log_data[17].valid := 1, [2055].log_data[18].valid := 1, [2055].log_data[19].valid := 1, [2055].time.Year := 2023, [2055].time.Month := 1, [2055].time.Day := 16, [2055].time.Hour := 19, [2055].time.Minute := 39, [2055].time.Second := 59, [2056].log_data[0].min := 1.0, [2056].log_data[0].max := 1.0, [2056].log_data[0].total := 300.0, [2056].log_data[0].time := 300.0, [2056].log_data[0].minminute := 40, [2056].log_data[0].maxminute := 40, [2056].log_data[0].valid := 1, [2056].log_data[1].valid := 1, [2056].log_data[2].valid := 1, [2056].log_data[3].valid := 1, [2056].log_data[4].valid := 1, [2056].log_data[5].valid := 1, [2056].log_data[6].valid := 1, [2056].log_data[7].valid := 1, [2056].log_data[8].valid := 1, [2056].log_data[9].valid := 1, [2056].log_data[10].valid := 1, [2056].log_data[11].valid := 1, [2056].log_data[12].valid := 1, [2056].log_data[13].valid := 1, [2056].log_data[14].valid := 1, [2056].log_data[15].valid := 1, [2056].log_data[16].valid := 1, [2056].log_data[17].valid := 1, [2056].log_data[18].valid := 1, [2056].log_data[19].valid := 1, [2056].time.Year := 2023, [2056].time.Month := 1, [2056].time.Day := 16, [2056].time.Hour := 19, [2056].time.Minute := 44, [2056].time.Second := 59, [2057].log_data[0].min := 1.0, [2057].log_data[0].max := 1.0, [2057].log_data[0].total := 300.0, [2057].log_data[0].time := 300.0,
        [2057].log_data[0].minminute := 45, [2057].log_data[0].maxminute := 45, [2057].log_data[0].valid := 1, [2057].log_data[1].valid := 1, [2057].log_data[2].valid := 1, [2057].log_data[3].valid := 1, [2057].log_data[4].valid := 1, [2057].log_data[5].valid := 1, [2057].log_data[6].valid := 1, [2057].log_data[7].valid := 1, [2057].log_data[8].valid := 1, [2057].log_data[9].valid := 1, [2057].log_data[10].valid := 1, [2057].log_data[11].valid := 1, [2057].log_data[12].valid := 1, [2057].log_data[13].valid := 1, [2057].log_data[14].valid := 1, [2057].log_data[15].valid := 1, [2057].log_data[16].valid := 1, [2057].log_data[17].valid := 1, [2057].log_data[18].valid := 1, [2057].log_data[19].valid := 1, [2057].time.Year := 2023, [2057].time.Month := 1, [2057].time.Day := 16, [2057].time.Hour := 19, [2057].time.Minute := 49, [2057].time.Second := 59, [2058].log_data[0].min := 1.0, [2058].log_data[0].max := 1.0, [2058].log_data[0].total := 300.0, [2058].log_data[0].time := 300.0, [2058].log_data[0].minminute := 50, [2058].log_data[0].maxminute := 50, [2058].log_data[0].valid := 1, [2058].log_data[1].valid := 1, [2058].log_data[2].valid := 1, [2058].log_data[3].valid := 1, [2058].log_data[4].valid := 1, [2058].log_data[5].valid := 1, [2058].log_data[6].valid := 1, [2058].log_data[7].valid := 1, [2058].log_data[8].valid := 1, [2058].log_data[9].valid := 1, [2058].log_data[10].valid := 1, [2058].log_data[11].valid := 1, [2058].log_data[12].valid := 1, [2058].log_data[13].valid := 1, [2058].log_data[14].valid := 1, [2058].log_data[15].valid := 1, [2058].log_data[16].valid := 1, [2058].log_data[17].valid := 1, [2058].log_data[18].valid := 1, [2058].log_data[19].valid := 1, [2058].time.Year := 2023, [2058].time.Month := 1, [2058].time.Day := 16, [2058].time.Hour := 19, [2058].time.Minute := 54, [2058].time.Second := 59,
        [2059].log_data[0].min := 1.0, [2059].log_data[0].max := 1.0, [2059].log_data[0].total := 300.0, [2059].log_data[0].time := 300.0, [2059].log_data[0].minminute := 55, [2059].log_data[0].maxminute := 55, [2059].log_data[0].valid := 1, [2059].log_data[1].valid := 1, [2059].log_data[2].valid := 1, [2059].log_data[3].valid := 1, [2059].log_data[4].valid := 1, [2059].log_data[5].valid := 1, [2059].log_data[6].valid := 1, [2059].log_data[7].valid := 1, [2059].log_data[8].valid := 1, [2059].log_data[9].valid := 1, [2059].log_data[10].valid := 1, [2059].log_data[11].valid := 1, [2059].log_data[12].valid := 1, [2059].log_data[13].valid := 1, [2059].log_data[14].valid := 1, [2059].log_data[15].valid := 1, [2059].log_data[16].valid := 1, [2059].log_data[17].valid := 1, [2059].log_data[18].valid := 1, [2059].log_data[19].valid := 1, [2059].time.Year := 2023, [2059].time.Month := 1, [2059].time.Day := 16, [2059].time.Hour := 19, [2059].time.Minute := 59, [2059].time.Second := 59, [2060].log_data[0].min := 1.0, [2060].log_data[0].max := 1.0, [2060].log_data[0].total := 300.0, [2060].log_data[0].time := 300.0, [2060].log_data[0].valid := 1, [2060].log_data[1].valid := 1, [2060].log_data[2].valid := 1, [2060].log_data[3].valid := 1, [2060].log_data[4].valid := 1, [2060].log_data[5].valid := 1, [2060].log_data[6].valid := 1, [2060].log_data[7].valid := 1, [2060].log_data[8].valid := 1, [2060].log_data[9].valid := 1, [2060].log_data[10].valid := 1, [2060].log_data[11].valid := 1, [2060].log_data[12].valid := 1, [2060].log_data[13].valid := 1, [2060].log_data[14].valid := 1, [2060].log_data[15].valid := 1, [2060].log_data[16].valid := 1, [2060].log_data[17].valid := 1, [2060].log_data[18].valid := 1, [2060].log_data[19].valid := 1, [2060].time.Year := 2023, [2060].time.Month := 1, [2060].time.Day := 16, [2060].time.Hour := 20,
        [2060].time.Minute := 4, [2060].time.Second := 59, [2061].log_data[0].min := 1.0, [2061].log_data[0].max := 1.0, [2061].log_data[0].total := 300.0, [2061].log_data[0].time := 300.0, [2061].log_data[0].minminute := 5, [2061].log_data[0].maxminute := 5, [2061].log_data[0].valid := 1, [2061].log_data[1].valid := 1, [2061].log_data[2].valid := 1, [2061].log_data[3].valid := 1, [2061].log_data[4].valid := 1, [2061].log_data[5].valid := 1, [2061].log_data[6].valid := 1, [2061].log_data[7].valid := 1, [2061].log_data[8].valid := 1, [2061].log_data[9].valid := 1, [2061].log_data[10].valid := 1, [2061].log_data[11].valid := 1, [2061].log_data[12].valid := 1, [2061].log_data[13].valid := 1, [2061].log_data[14].valid := 1, [2061].log_data[15].valid := 1, [2061].log_data[16].valid := 1, [2061].log_data[17].valid := 1, [2061].log_data[18].valid := 1, [2061].log_data[19].valid := 1, [2061].time.Year := 2023, [2061].time.Month := 1, [2061].time.Day := 16, [2061].time.Hour := 20, [2061].time.Minute := 9, [2061].time.Second := 59, [2062].log_data[0].min := 1.0, [2062].log_data[0].max := 1.0, [2062].log_data[0].total := 300.0, [2062].log_data[0].time := 300.0, [2062].log_data[0].minminute := 10, [2062].log_data[0].maxminute := 10, [2062].log_data[0].valid := 1, [2062].log_data[1].valid := 1, [2062].log_data[2].valid := 1, [2062].log_data[3].valid := 1, [2062].log_data[4].valid := 1, [2062].log_data[5].valid := 1, [2062].log_data[6].valid := 1, [2062].log_data[7].valid := 1, [2062].log_data[8].valid := 1, [2062].log_data[9].valid := 1, [2062].log_data[10].valid := 1, [2062].log_data[11].valid := 1, [2062].log_data[12].valid := 1, [2062].log_data[13].valid := 1, [2062].log_data[14].valid := 1, [2062].log_data[15].valid := 1, [2062].log_data[16].valid := 1, [2062].log_data[17].valid := 1, [2062].log_data[18].valid := 1, [2062].log_data[19].valid := 1,
        [2062].time.Year := 2023, [2062].time.Month := 1, [2062].time.Day := 16, [2062].time.Hour := 20, [2062].time.Minute := 14, [2062].time.Second := 59, [2063].log_data[0].min := 1.0, [2063].log_data[0].max := 1.0, [2063].log_data[0].total := 300.0, [2063].log_data[0].time := 300.0, [2063].log_data[0].minminute := 15, [2063].log_data[0].maxminute := 15, [2063].log_data[0].valid := 1, [2063].log_data[1].valid := 1, [2063].log_data[2].valid := 1, [2063].log_data[3].valid := 1, [2063].log_data[4].valid := 1, [2063].log_data[5].valid := 1, [2063].log_data[6].valid := 1, [2063].log_data[7].valid := 1, [2063].log_data[8].valid := 1, [2063].log_data[9].valid := 1, [2063].log_data[10].valid := 1, [2063].log_data[11].valid := 1, [2063].log_data[12].valid := 1, [2063].log_data[13].valid := 1, [2063].log_data[14].valid := 1, [2063].log_data[15].valid := 1, [2063].log_data[16].valid := 1, [2063].log_data[17].valid := 1, [2063].log_data[18].valid := 1, [2063].log_data[19].valid := 1, [2063].time.Year := 2023, [2063].time.Month := 1, [2063].time.Day := 16, [2063].time.Hour := 20, [2063].time.Minute := 19, [2063].time.Second := 59, [2064].log_data[0].min := 1.0, [2064].log_data[0].max := 1.0, [2064].log_data[0].total := 300.0, [2064].log_data[0].time := 300.0, [2064].log_data[0].minminute := 20, [2064].log_data[0].maxminute := 20, [2064].log_data[0].valid := 1, [2064].log_data[1].valid := 1, [2064].log_data[2].valid := 1, [2064].log_data[3].valid := 1, [2064].log_data[4].valid := 1, [2064].log_data[5].valid := 1, [2064].log_data[6].valid := 1, [2064].log_data[7].valid := 1, [2064].log_data[8].valid := 1, [2064].log_data[9].valid := 1, [2064].log_data[10].valid := 1, [2064].log_data[11].valid := 1, [2064].log_data[12].valid := 1, [2064].log_data[13].valid := 1, [2064].log_data[14].valid := 1, [2064].log_data[15].valid := 1,
        [2064].log_data[16].valid := 1, [2064].log_data[17].valid := 1, [2064].log_data[18].valid := 1, [2064].log_data[19].valid := 1, [2064].time.Year := 2023, [2064].time.Month := 1, [2064].time.Day := 16, [2064].time.Hour := 20, [2064].time.Minute := 24, [2064].time.Second := 59, [2065].log_data[0].min := 1.0, [2065].log_data[0].max := 1.0, [2065].log_data[0].total := 300.0, [2065].log_data[0].time := 300.0, [2065].log_data[0].minminute := 25, [2065].log_data[0].maxminute := 25, [2065].log_data[0].valid := 1, [2065].log_data[1].valid := 1, [2065].log_data[2].valid := 1, [2065].log_data[3].valid := 1, [2065].log_data[4].valid := 1, [2065].log_data[5].valid := 1, [2065].log_data[6].valid := 1, [2065].log_data[7].valid := 1, [2065].log_data[8].valid := 1, [2065].log_data[9].valid := 1, [2065].log_data[10].valid := 1, [2065].log_data[11].valid := 1, [2065].log_data[12].valid := 1, [2065].log_data[13].valid := 1, [2065].log_data[14].valid := 1, [2065].log_data[15].valid := 1, [2065].log_data[16].valid := 1, [2065].log_data[17].valid := 1, [2065].log_data[18].valid := 1, [2065].log_data[19].valid := 1, [2065].time.Year := 2023, [2065].time.Month := 1, [2065].time.Day := 16, [2065].time.Hour := 20, [2065].time.Minute := 29, [2065].time.Second := 59, [2066].log_data[0].min := 1.0, [2066].log_data[0].max := 1.0, [2066].log_data[0].total := 300.0, [2066].log_data[0].time := 300.0, [2066].log_data[0].minminute := 30, [2066].log_data[0].maxminute := 30, [2066].log_data[0].valid := 1, [2066].log_data[1].valid := 1, [2066].log_data[2].valid := 1, [2066].log_data[3].valid := 1, [2066].log_data[4].valid := 1, [2066].log_data[5].valid := 1, [2066].log_data[6].valid := 1, [2066].log_data[7].valid := 1, [2066].log_data[8].valid := 1, [2066].log_data[9].valid := 1, [2066].log_data[10].valid := 1, [2066].log_data[11].valid := 1,
        [2066].log_data[12].valid := 1, [2066].log_data[13].valid := 1, [2066].log_data[14].valid := 1, [2066].log_data[15].valid := 1, [2066].log_data[16].valid := 1, [2066].log_data[17].valid := 1, [2066].log_data[18].valid := 1, [2066].log_data[19].valid := 1, [2066].time.Year := 2023, [2066].time.Month := 1, [2066].time.Day := 16, [2066].time.Hour := 20, [2066].time.Minute := 34, [2066].time.Second := 59, [2067].log_data[0].min := 1.0, [2067].log_data[0].max := 1.0, [2067].log_data[0].total := 300.0, [2067].log_data[0].time := 300.0, [2067].log_data[0].minminute := 35, [2067].log_data[0].maxminute := 35, [2067].log_data[0].valid := 1, [2067].log_data[1].valid := 1, [2067].log_data[2].valid := 1, [2067].log_data[3].valid := 1, [2067].log_data[4].valid := 1, [2067].log_data[5].valid := 1, [2067].log_data[6].valid := 1, [2067].log_data[7].valid := 1, [2067].log_data[8].valid := 1, [2067].log_data[9].valid := 1, [2067].log_data[10].valid := 1, [2067].log_data[11].valid := 1, [2067].log_data[12].valid := 1, [2067].log_data[13].valid := 1, [2067].log_data[14].valid := 1, [2067].log_data[15].valid := 1, [2067].log_data[16].valid := 1, [2067].log_data[17].valid := 1, [2067].log_data[18].valid := 1, [2067].log_data[19].valid := 1, [2067].time.Year := 2023, [2067].time.Month := 1, [2067].time.Day := 16, [2067].time.Hour := 20, [2067].time.Minute := 39, [2067].time.Second := 59, [2068].log_data[0].min := 1.0, [2068].log_data[0].max := 1.0, [2068].log_data[0].total := 300.0, [2068].log_data[0].time := 300.0, [2068].log_data[0].minminute := 40, [2068].log_data[0].maxminute := 40, [2068].log_data[0].valid := 1, [2068].log_data[1].valid := 1, [2068].log_data[2].valid := 1, [2068].log_data[3].valid := 1, [2068].log_data[4].valid := 1, [2068].log_data[5].valid := 1, [2068].log_data[6].valid := 1, [2068].log_data[7].valid := 1,
        [2068].log_data[8].valid := 1, [2068].log_data[9].valid := 1, [2068].log_data[10].valid := 1, [2068].log_data[11].valid := 1, [2068].log_data[12].valid := 1, [2068].log_data[13].valid := 1, [2068].log_data[14].valid := 1, [2068].log_data[15].valid := 1, [2068].log_data[16].valid := 1, [2068].log_data[17].valid := 1, [2068].log_data[18].valid := 1, [2068].log_data[19].valid := 1, [2068].time.Year := 2023, [2068].time.Month := 1, [2068].time.Day := 16, [2068].time.Hour := 20, [2068].time.Minute := 44, [2068].time.Second := 59, [2069].log_data[0].min := 1.0, [2069].log_data[0].max := 1.0, [2069].log_data[0].total := 300.0, [2069].log_data[0].time := 300.0, [2069].log_data[0].minminute := 45, [2069].log_data[0].maxminute := 45, [2069].log_data[0].valid := 1, [2069].log_data[1].valid := 1, [2069].log_data[2].valid := 1, [2069].log_data[3].valid := 1, [2069].log_data[4].valid := 1, [2069].log_data[5].valid := 1, [2069].log_data[6].valid := 1, [2069].log_data[7].valid := 1, [2069].log_data[8].valid := 1, [2069].log_data[9].valid := 1, [2069].log_data[10].valid := 1, [2069].log_data[11].valid := 1, [2069].log_data[12].valid := 1, [2069].log_data[13].valid := 1, [2069].log_data[14].valid := 1, [2069].log_data[15].valid := 1, [2069].log_data[16].valid := 1, [2069].log_data[17].valid := 1, [2069].log_data[18].valid := 1, [2069].log_data[19].valid := 1, [2069].time.Year := 2023, [2069].time.Month := 1, [2069].time.Day := 16, [2069].time.Hour := 20, [2069].time.Minute := 49, [2069].time.Second := 59, [2070].log_data[0].min := 1.0, [2070].log_data[0].max := 1.0, [2070].log_data[0].total := 300.0, [2070].log_data[0].time := 300.0, [2070].log_data[0].minminute := 50, [2070].log_data[0].maxminute := 50, [2070].log_data[0].valid := 1, [2070].log_data[1].valid := 1, [2070].log_data[2].valid := 1, [2070].log_data[3].valid := 1,
        [2070].log_data[4].valid := 1, [2070].log_data[5].valid := 1, [2070].log_data[6].valid := 1, [2070].log_data[7].valid := 1, [2070].log_data[8].valid := 1, [2070].log_data[9].valid := 1, [2070].log_data[10].valid := 1, [2070].log_data[11].valid := 1, [2070].log_data[12].valid := 1, [2070].log_data[13].valid := 1, [2070].log_data[14].valid := 1, [2070].log_data[15].valid := 1, [2070].log_data[16].valid := 1, [2070].log_data[17].valid := 1, [2070].log_data[18].valid := 1, [2070].log_data[19].valid := 1, [2070].time.Year := 2023, [2070].time.Month := 1, [2070].time.Day := 16, [2070].time.Hour := 20, [2070].time.Minute := 54, [2070].time.Second := 59, [2071].log_data[0].min := 1.0, [2071].log_data[0].max := 1.0, [2071].log_data[0].total := 300.0, [2071].log_data[0].time := 300.0, [2071].log_data[0].minminute := 55, [2071].log_data[0].maxminute := 55, [2071].log_data[0].valid := 1, [2071].log_data[1].valid := 1, [2071].log_data[2].valid := 1, [2071].log_data[3].valid := 1, [2071].log_data[4].valid := 1, [2071].log_data[5].valid := 1, [2071].log_data[6].valid := 1, [2071].log_data[7].valid := 1, [2071].log_data[8].valid := 1, [2071].log_data[9].valid := 1, [2071].log_data[10].valid := 1, [2071].log_data[11].valid := 1, [2071].log_data[12].valid := 1, [2071].log_data[13].valid := 1, [2071].log_data[14].valid := 1, [2071].log_data[15].valid := 1, [2071].log_data[16].valid := 1, [2071].log_data[17].valid := 1, [2071].log_data[18].valid := 1, [2071].log_data[19].valid := 1, [2071].time.Year := 2023, [2071].time.Month := 1, [2071].time.Day := 16, [2071].time.Hour := 20, [2071].time.Minute := 59, [2071].time.Second := 59, [2072].log_data[0].min := 1.0, [2072].log_data[0].max := 1.0, [2072].log_data[0].total := 299.5, [2072].log_data[0].time := 299.5, [2072].log_data[0].valid := 1, [2072].log_data[1].valid := 1,
        [2072].log_data[2].valid := 1, [2072].log_data[3].valid := 1, [2072].log_data[4].valid := 1, [2072].log_data[5].valid := 1, [2072].log_data[6].valid := 1, [2072].log_data[7].valid := 1, [2072].log_data[8].valid := 1, [2072].log_data[9].valid := 1, [2072].log_data[10].valid := 1, [2072].log_data[11].valid := 1, [2072].log_data[12].valid := 1, [2072].log_data[13].valid := 1, [2072].log_data[14].valid := 1, [2072].log_data[15].valid := 1, [2072].log_data[16].valid := 1, [2072].log_data[17].valid := 1, [2072].log_data[18].valid := 1, [2072].log_data[19].valid := 1, [2072].time.Year := 2023, [2072].time.Month := 1, [2072].time.Day := 16, [2072].time.Hour := 21, [2072].time.Minute := 4, [2072].time.Second := 59, [2073].log_data[0].min := 1.0, [2073].log_data[0].max := 1.0, [2073].log_data[0].total := 300.0, [2073].log_data[0].time := 300.0, [2073].log_data[0].minminute := 5, [2073].log_data[0].maxminute := 5, [2073].log_data[0].valid := 1, [2073].log_data[1].valid := 1, [2073].log_data[2].valid := 1, [2073].log_data[3].valid := 1, [2073].log_data[4].valid := 1, [2073].log_data[5].valid := 1, [2073].log_data[6].valid := 1, [2073].log_data[7].valid := 1, [2073].log_data[8].valid := 1, [2073].log_data[9].valid := 1, [2073].log_data[10].valid := 1, [2073].log_data[11].valid := 1, [2073].log_data[12].valid := 1, [2073].log_data[13].valid := 1, [2073].log_data[14].valid := 1, [2073].log_data[15].valid := 1, [2073].log_data[16].valid := 1, [2073].log_data[17].valid := 1, [2073].log_data[18].valid := 1, [2073].log_data[19].valid := 1, [2073].time.Year := 2023, [2073].time.Month := 1, [2073].time.Day := 16, [2073].time.Hour := 21, [2073].time.Minute := 9, [2073].time.Second := 59, [2074].log_data[0].min := 1.0, [2074].log_data[0].max := 1.0, [2074].log_data[0].total := 300.0, [2074].log_data[0].time := 300.0,
        [2074].log_data[0].minminute := 10, [2074].log_data[0].maxminute := 10, [2074].log_data[0].valid := 1, [2074].log_data[1].valid := 1, [2074].log_data[2].valid := 1, [2074].log_data[3].valid := 1, [2074].log_data[4].valid := 1, [2074].log_data[5].valid := 1, [2074].log_data[6].valid := 1, [2074].log_data[7].valid := 1, [2074].log_data[8].valid := 1, [2074].log_data[9].valid := 1, [2074].log_data[10].valid := 1, [2074].log_data[11].valid := 1, [2074].log_data[12].valid := 1, [2074].log_data[13].valid := 1, [2074].log_data[14].valid := 1, [2074].log_data[15].valid := 1, [2074].log_data[16].valid := 1, [2074].log_data[17].valid := 1, [2074].log_data[18].valid := 1, [2074].log_data[19].valid := 1, [2074].time.Year := 2023, [2074].time.Month := 1, [2074].time.Day := 16, [2074].time.Hour := 21, [2074].time.Minute := 14, [2074].time.Second := 59, [2075].log_data[0].min := 1.0, [2075].log_data[0].max := 1.0, [2075].log_data[0].total := 300.0, [2075].log_data[0].time := 300.0, [2075].log_data[0].minminute := 15, [2075].log_data[0].maxminute := 15, [2075].log_data[0].valid := 1, [2075].log_data[1].valid := 1, [2075].log_data[2].valid := 1, [2075].log_data[3].valid := 1, [2075].log_data[4].valid := 1, [2075].log_data[5].valid := 1, [2075].log_data[6].valid := 1, [2075].log_data[7].valid := 1, [2075].log_data[8].valid := 1, [2075].log_data[9].valid := 1, [2075].log_data[10].valid := 1, [2075].log_data[11].valid := 1, [2075].log_data[12].valid := 1, [2075].log_data[13].valid := 1, [2075].log_data[14].valid := 1, [2075].log_data[15].valid := 1, [2075].log_data[16].valid := 1, [2075].log_data[17].valid := 1, [2075].log_data[18].valid := 1, [2075].log_data[19].valid := 1, [2075].time.Year := 2023, [2075].time.Month := 1, [2075].time.Day := 16, [2075].time.Hour := 21, [2075].time.Minute := 19, [2075].time.Second := 59,
        [2076].log_data[0].min := 1.0, [2076].log_data[0].max := 1.0, [2076].log_data[0].total := 300.0, [2076].log_data[0].time := 300.0, [2076].log_data[0].minminute := 20, [2076].log_data[0].maxminute := 20, [2076].log_data[0].valid := 1, [2076].log_data[1].valid := 1, [2076].log_data[2].valid := 1, [2076].log_data[3].valid := 1, [2076].log_data[4].valid := 1, [2076].log_data[5].valid := 1, [2076].log_data[6].valid := 1, [2076].log_data[7].valid := 1, [2076].log_data[8].valid := 1, [2076].log_data[9].valid := 1, [2076].log_data[10].valid := 1, [2076].log_data[11].valid := 1, [2076].log_data[12].valid := 1, [2076].log_data[13].valid := 1, [2076].log_data[14].valid := 1, [2076].log_data[15].valid := 1, [2076].log_data[16].valid := 1, [2076].log_data[17].valid := 1, [2076].log_data[18].valid := 1, [2076].log_data[19].valid := 1, [2076].time.Year := 2023, [2076].time.Month := 1, [2076].time.Day := 16, [2076].time.Hour := 21, [2076].time.Minute := 24, [2076].time.Second := 59, [2077].log_data[0].min := 1.0, [2077].log_data[0].max := 1.0, [2077].log_data[0].total := 300.0, [2077].log_data[0].time := 300.0, [2077].log_data[0].minminute := 25, [2077].log_data[0].maxminute := 25, [2077].log_data[0].valid := 1, [2077].log_data[1].valid := 1, [2077].log_data[2].valid := 1, [2077].log_data[3].valid := 1, [2077].log_data[4].valid := 1, [2077].log_data[5].valid := 1, [2077].log_data[6].valid := 1, [2077].log_data[7].valid := 1, [2077].log_data[8].valid := 1, [2077].log_data[9].valid := 1, [2077].log_data[10].valid := 1, [2077].log_data[11].valid := 1, [2077].log_data[12].valid := 1, [2077].log_data[13].valid := 1, [2077].log_data[14].valid := 1, [2077].log_data[15].valid := 1, [2077].log_data[16].valid := 1, [2077].log_data[17].valid := 1, [2077].log_data[18].valid := 1, [2077].log_data[19].valid := 1, [2077].time.Year := 2023, [2077].time.Month := 1,
        [2077].time.Day := 16, [2077].time.Hour := 21, [2077].time.Minute := 29, [2077].time.Second := 59, [2078].log_data[0].min := 1.0, [2078].log_data[0].max := 1.0, [2078].log_data[0].total := 300.0, [2078].log_data[0].time := 300.0, [2078].log_data[0].minminute := 30, [2078].log_data[0].maxminute := 30, [2078].log_data[0].valid := 1, [2078].log_data[1].valid := 1, [2078].log_data[2].valid := 1, [2078].log_data[3].valid := 1, [2078].log_data[4].valid := 1, [2078].log_data[5].valid := 1, [2078].log_data[6].valid := 1, [2078].log_data[7].valid := 1, [2078].log_data[8].valid := 1, [2078].log_data[9].valid := 1, [2078].log_data[10].valid := 1, [2078].log_data[11].valid := 1, [2078].log_data[12].valid := 1, [2078].log_data[13].valid := 1, [2078].log_data[14].valid := 1, [2078].log_data[15].valid := 1, [2078].log_data[16].valid := 1, [2078].log_data[17].valid := 1, [2078].log_data[18].valid := 1, [2078].log_data[19].valid := 1, [2078].time.Year := 2023, [2078].time.Month := 1, [2078].time.Day := 16, [2078].time.Hour := 21, [2078].time.Minute := 34, [2078].time.Second := 59, [2079].log_data[0].min := 1.0, [2079].log_data[0].max := 1.0, [2079].log_data[0].total := 300.0, [2079].log_data[0].time := 300.0, [2079].log_data[0].minminute := 35, [2079].log_data[0].maxminute := 35, [2079].log_data[0].valid := 1, [2079].log_data[1].valid := 1, [2079].log_data[2].valid := 1, [2079].log_data[3].valid := 1, [2079].log_data[4].valid := 1, [2079].log_data[5].valid := 1, [2079].log_data[6].valid := 1, [2079].log_data[7].valid := 1, [2079].log_data[8].valid := 1, [2079].log_data[9].valid := 1, [2079].log_data[10].valid := 1, [2079].log_data[11].valid := 1, [2079].log_data[12].valid := 1, [2079].log_data[13].valid := 1, [2079].log_data[14].valid := 1, [2079].log_data[15].valid := 1, [2079].log_data[16].valid := 1, [2079].log_data[17].valid := 1,
        [2079].log_data[18].valid := 1, [2079].log_data[19].valid := 1, [2079].time.Year := 2023, [2079].time.Month := 1, [2079].time.Day := 16, [2079].time.Hour := 21, [2079].time.Minute := 39, [2079].time.Second := 59, [2080].log_data[0].min := 1.0, [2080].log_data[0].max := 1.0, [2080].log_data[0].total := 300.0, [2080].log_data[0].time := 300.0, [2080].log_data[0].minminute := 40, [2080].log_data[0].maxminute := 40, [2080].log_data[0].valid := 1, [2080].log_data[1].valid := 1, [2080].log_data[2].valid := 1, [2080].log_data[3].valid := 1, [2080].log_data[4].valid := 1, [2080].log_data[5].valid := 1, [2080].log_data[6].valid := 1, [2080].log_data[7].valid := 1, [2080].log_data[8].valid := 1, [2080].log_data[9].valid := 1, [2080].log_data[10].valid := 1, [2080].log_data[11].valid := 1, [2080].log_data[12].valid := 1, [2080].log_data[13].valid := 1, [2080].log_data[14].valid := 1, [2080].log_data[15].valid := 1, [2080].log_data[16].valid := 1, [2080].log_data[17].valid := 1, [2080].log_data[18].valid := 1, [2080].log_data[19].valid := 1, [2080].time.Year := 2023, [2080].time.Month := 1, [2080].time.Day := 16, [2080].time.Hour := 21, [2080].time.Minute := 44, [2080].time.Second := 59, [2081].log_data[0].min := 1.0, [2081].log_data[0].max := 1.0, [2081].log_data[0].total := 300.0, [2081].log_data[0].time := 300.0, [2081].log_data[0].minminute := 45, [2081].log_data[0].maxminute := 45, [2081].log_data[0].valid := 1, [2081].log_data[1].valid := 1, [2081].log_data[2].valid := 1, [2081].log_data[3].valid := 1, [2081].log_data[4].valid := 1, [2081].log_data[5].valid := 1, [2081].log_data[6].valid := 1, [2081].log_data[7].valid := 1, [2081].log_data[8].valid := 1, [2081].log_data[9].valid := 1, [2081].log_data[10].valid := 1, [2081].log_data[11].valid := 1, [2081].log_data[12].valid := 1, [2081].log_data[13].valid := 1,
        [2081].log_data[14].valid := 1, [2081].log_data[15].valid := 1, [2081].log_data[16].valid := 1, [2081].log_data[17].valid := 1, [2081].log_data[18].valid := 1, [2081].log_data[19].valid := 1, [2081].time.Year := 2023, [2081].time.Month := 1, [2081].time.Day := 16, [2081].time.Hour := 21, [2081].time.Minute := 49, [2081].time.Second := 59, [2082].log_data[0].min := 1.0, [2082].log_data[0].max := 1.0, [2082].log_data[0].total := 300.0, [2082].log_data[0].time := 300.0, [2082].log_data[0].minminute := 50, [2082].log_data[0].maxminute := 50, [2082].log_data[0].valid := 1, [2082].log_data[1].valid := 1, [2082].log_data[2].valid := 1, [2082].log_data[3].valid := 1, [2082].log_data[4].valid := 1, [2082].log_data[5].valid := 1, [2082].log_data[6].valid := 1, [2082].log_data[7].valid := 1, [2082].log_data[8].valid := 1, [2082].log_data[9].valid := 1, [2082].log_data[10].valid := 1, [2082].log_data[11].valid := 1, [2082].log_data[12].valid := 1, [2082].log_data[13].valid := 1, [2082].log_data[14].valid := 1, [2082].log_data[15].valid := 1, [2082].log_data[16].valid := 1, [2082].log_data[17].valid := 1, [2082].log_data[18].valid := 1, [2082].log_data[19].valid := 1, [2082].time.Year := 2023, [2082].time.Month := 1, [2082].time.Day := 16, [2082].time.Hour := 21, [2082].time.Minute := 54, [2082].time.Second := 59, [2083].log_data[0].min := 1.0, [2083].log_data[0].max := 1.0, [2083].log_data[0].total := 300.0, [2083].log_data[0].time := 300.0, [2083].log_data[0].minminute := 55, [2083].log_data[0].maxminute := 55, [2083].log_data[0].valid := 1, [2083].log_data[1].valid := 1, [2083].log_data[2].valid := 1, [2083].log_data[3].valid := 1, [2083].log_data[4].valid := 1, [2083].log_data[5].valid := 1, [2083].log_data[6].valid := 1, [2083].log_data[7].valid := 1, [2083].log_data[8].valid := 1, [2083].log_data[9].valid := 1,
        [2083].log_data[10].valid := 1, [2083].log_data[11].valid := 1, [2083].log_data[12].valid := 1, [2083].log_data[13].valid := 1, [2083].log_data[14].valid := 1, [2083].log_data[15].valid := 1, [2083].log_data[16].valid := 1, [2083].log_data[17].valid := 1, [2083].log_data[18].valid := 1, [2083].log_data[19].valid := 1, [2083].time.Year := 2023, [2083].time.Month := 1, [2083].time.Day := 16, [2083].time.Hour := 21, [2083].time.Minute := 59, [2083].time.Second := 59, [2084].log_data[0].min := 1.0, [2084].log_data[0].max := 1.0, [2084].log_data[0].total := 300.0, [2084].log_data[0].time := 300.0, [2084].log_data[0].valid := 1, [2084].log_data[1].valid := 1, [2084].log_data[2].valid := 1, [2084].log_data[3].valid := 1, [2084].log_data[4].valid := 1, [2084].log_data[5].valid := 1, [2084].log_data[6].valid := 1, [2084].log_data[7].valid := 1, [2084].log_data[8].valid := 1, [2084].log_data[9].valid := 1, [2084].log_data[10].valid := 1, [2084].log_data[11].valid := 1, [2084].log_data[12].valid := 1, [2084].log_data[13].valid := 1, [2084].log_data[14].valid := 1, [2084].log_data[15].valid := 1, [2084].log_data[16].valid := 1, [2084].log_data[17].valid := 1, [2084].log_data[18].valid := 1, [2084].log_data[19].valid := 1, [2084].time.Year := 2023, [2084].time.Month := 1, [2084].time.Day := 16, [2084].time.Hour := 22, [2084].time.Minute := 4, [2084].time.Second := 59, [2085].log_data[0].min := 1.0, [2085].log_data[0].max := 1.0, [2085].log_data[0].total := 300.0, [2085].log_data[0].time := 300.0, [2085].log_data[0].minminute := 5, [2085].log_data[0].maxminute := 5, [2085].log_data[0].valid := 1, [2085].log_data[1].valid := 1, [2085].log_data[2].valid := 1, [2085].log_data[3].valid := 1, [2085].log_data[4].valid := 1, [2085].log_data[5].valid := 1, [2085].log_data[6].valid := 1, [2085].log_data[7].valid := 1,
        [2085].log_data[8].valid := 1, [2085].log_data[9].valid := 1, [2085].log_data[10].valid := 1, [2085].log_data[11].valid := 1, [2085].log_data[12].valid := 1, [2085].log_data[13].valid := 1, [2085].log_data[14].valid := 1, [2085].log_data[15].valid := 1, [2085].log_data[16].valid := 1, [2085].log_data[17].valid := 1, [2085].log_data[18].valid := 1, [2085].log_data[19].valid := 1, [2085].time.Year := 2023, [2085].time.Month := 1, [2085].time.Day := 16, [2085].time.Hour := 22, [2085].time.Minute := 9, [2085].time.Second := 59, [2086].log_data[0].min := 1.0, [2086].log_data[0].max := 1.0, [2086].log_data[0].total := 300.0, [2086].log_data[0].time := 300.0, [2086].log_data[0].minminute := 10, [2086].log_data[0].maxminute := 10, [2086].log_data[0].valid := 1, [2086].log_data[1].valid := 1, [2086].log_data[2].valid := 1, [2086].log_data[3].valid := 1, [2086].log_data[4].valid := 1, [2086].log_data[5].valid := 1, [2086].log_data[6].valid := 1, [2086].log_data[7].valid := 1, [2086].log_data[8].valid := 1, [2086].log_data[9].valid := 1, [2086].log_data[10].valid := 1, [2086].log_data[11].valid := 1, [2086].log_data[12].valid := 1, [2086].log_data[13].valid := 1, [2086].log_data[14].valid := 1, [2086].log_data[15].valid := 1, [2086].log_data[16].valid := 1, [2086].log_data[17].valid := 1, [2086].log_data[18].valid := 1, [2086].log_data[19].valid := 1, [2086].time.Year := 2023, [2086].time.Month := 1, [2086].time.Day := 16, [2086].time.Hour := 22, [2086].time.Minute := 14, [2086].time.Second := 59, [2087].log_data[0].min := 1.0, [2087].log_data[0].max := 1.0, [2087].log_data[0].total := 300.0, [2087].log_data[0].time := 300.0, [2087].log_data[0].minminute := 15, [2087].log_data[0].maxminute := 15, [2087].log_data[0].valid := 1, [2087].log_data[1].valid := 1, [2087].log_data[2].valid := 1, [2087].log_data[3].valid := 1,
        [2087].log_data[4].valid := 1, [2087].log_data[5].valid := 1, [2087].log_data[6].valid := 1, [2087].log_data[7].valid := 1, [2087].log_data[8].valid := 1, [2087].log_data[9].valid := 1, [2087].log_data[10].valid := 1, [2087].log_data[11].valid := 1, [2087].log_data[12].valid := 1, [2087].log_data[13].valid := 1, [2087].log_data[14].valid := 1, [2087].log_data[15].valid := 1, [2087].log_data[16].valid := 1, [2087].log_data[17].valid := 1, [2087].log_data[18].valid := 1, [2087].log_data[19].valid := 1, [2087].time.Year := 2023, [2087].time.Month := 1, [2087].time.Day := 16, [2087].time.Hour := 22, [2087].time.Minute := 19, [2087].time.Second := 59, [2088].log_data[0].min := 1.0, [2088].log_data[0].max := 1.0, [2088].log_data[0].total := 300.0, [2088].log_data[0].time := 300.0, [2088].log_data[0].minminute := 20, [2088].log_data[0].maxminute := 20, [2088].log_data[0].valid := 1, [2088].log_data[1].valid := 1, [2088].log_data[2].valid := 1, [2088].log_data[3].valid := 1, [2088].log_data[4].valid := 1, [2088].log_data[5].valid := 1, [2088].log_data[6].valid := 1, [2088].log_data[7].valid := 1, [2088].log_data[8].valid := 1, [2088].log_data[9].valid := 1, [2088].log_data[10].valid := 1, [2088].log_data[11].valid := 1, [2088].log_data[12].valid := 1, [2088].log_data[13].valid := 1, [2088].log_data[14].valid := 1, [2088].log_data[15].valid := 1, [2088].log_data[16].valid := 1, [2088].log_data[17].valid := 1, [2088].log_data[18].valid := 1, [2088].log_data[19].valid := 1, [2088].time.Year := 2023, [2088].time.Month := 1, [2088].time.Day := 16, [2088].time.Hour := 22, [2088].time.Minute := 24, [2088].time.Second := 59, [2089].log_data[0].min := 1.0, [2089].log_data[0].max := 1.0, [2089].log_data[0].total := 300.0, [2089].log_data[0].time := 300.0, [2089].log_data[0].minminute := 25, [2089].log_data[0].maxminute := 25,
        [2089].log_data[0].valid := 1, [2089].log_data[1].valid := 1, [2089].log_data[2].valid := 1, [2089].log_data[3].valid := 1, [2089].log_data[4].valid := 1, [2089].log_data[5].valid := 1, [2089].log_data[6].valid := 1, [2089].log_data[7].valid := 1, [2089].log_data[8].valid := 1, [2089].log_data[9].valid := 1, [2089].log_data[10].valid := 1, [2089].log_data[11].valid := 1, [2089].log_data[12].valid := 1, [2089].log_data[13].valid := 1, [2089].log_data[14].valid := 1, [2089].log_data[15].valid := 1, [2089].log_data[16].valid := 1, [2089].log_data[17].valid := 1, [2089].log_data[18].valid := 1, [2089].log_data[19].valid := 1, [2089].time.Year := 2023, [2089].time.Month := 1, [2089].time.Day := 16, [2089].time.Hour := 22, [2089].time.Minute := 29, [2089].time.Second := 59, [2090].log_data[0].min := 1.0, [2090].log_data[0].max := 1.0, [2090].log_data[0].total := 300.0, [2090].log_data[0].time := 300.0, [2090].log_data[0].minminute := 30, [2090].log_data[0].maxminute := 30, [2090].log_data[0].valid := 1, [2090].log_data[1].valid := 1, [2090].log_data[2].valid := 1, [2090].log_data[3].valid := 1, [2090].log_data[4].valid := 1, [2090].log_data[5].valid := 1, [2090].log_data[6].valid := 1, [2090].log_data[7].valid := 1, [2090].log_data[8].valid := 1, [2090].log_data[9].valid := 1, [2090].log_data[10].valid := 1, [2090].log_data[11].valid := 1, [2090].log_data[12].valid := 1, [2090].log_data[13].valid := 1, [2090].log_data[14].valid := 1, [2090].log_data[15].valid := 1, [2090].log_data[16].valid := 1, [2090].log_data[17].valid := 1, [2090].log_data[18].valid := 1, [2090].log_data[19].valid := 1, [2090].time.Year := 2023, [2090].time.Month := 1, [2090].time.Day := 16, [2090].time.Hour := 22, [2090].time.Minute := 34, [2090].time.Second := 59, [2091].log_data[0].min := 1.0, [2091].log_data[0].max := 1.0,
        [2091].log_data[0].total := 300.0, [2091].log_data[0].time := 300.0, [2091].log_data[0].minminute := 35, [2091].log_data[0].maxminute := 35, [2091].log_data[0].valid := 1, [2091].log_data[1].valid := 1, [2091].log_data[2].valid := 1, [2091].log_data[3].valid := 1, [2091].log_data[4].valid := 1, [2091].log_data[5].valid := 1, [2091].log_data[6].valid := 1, [2091].log_data[7].valid := 1, [2091].log_data[8].valid := 1, [2091].log_data[9].valid := 1, [2091].log_data[10].valid := 1, [2091].log_data[11].valid := 1, [2091].log_data[12].valid := 1, [2091].log_data[13].valid := 1, [2091].log_data[14].valid := 1, [2091].log_data[15].valid := 1, [2091].log_data[16].valid := 1, [2091].log_data[17].valid := 1, [2091].log_data[18].valid := 1, [2091].log_data[19].valid := 1, [2091].time.Year := 2023, [2091].time.Month := 1, [2091].time.Day := 16, [2091].time.Hour := 22, [2091].time.Minute := 39, [2091].time.Second := 59, [2092].log_data[0].min := 1.0, [2092].log_data[0].max := 1.0, [2092].log_data[0].total := 300.0, [2092].log_data[0].time := 300.0, [2092].log_data[0].minminute := 40, [2092].log_data[0].maxminute := 40, [2092].log_data[0].valid := 1, [2092].log_data[1].valid := 1, [2092].log_data[2].valid := 1, [2092].log_data[3].valid := 1, [2092].log_data[4].valid := 1, [2092].log_data[5].valid := 1, [2092].log_data[6].valid := 1, [2092].log_data[7].valid := 1, [2092].log_data[8].valid := 1, [2092].log_data[9].valid := 1, [2092].log_data[10].valid := 1, [2092].log_data[11].valid := 1, [2092].log_data[12].valid := 1, [2092].log_data[13].valid := 1, [2092].log_data[14].valid := 1, [2092].log_data[15].valid := 1, [2092].log_data[16].valid := 1, [2092].log_data[17].valid := 1, [2092].log_data[18].valid := 1, [2092].log_data[19].valid := 1, [2092].time.Year := 2023, [2092].time.Month := 1, [2092].time.Day := 16, [2092].time.Hour := 22,
        [2092].time.Minute := 44, [2092].time.Second := 59, [2093].log_data[0].min := 1.0, [2093].log_data[0].max := 1.0, [2093].log_data[0].total := 300.0, [2093].log_data[0].time := 300.0, [2093].log_data[0].minminute := 45, [2093].log_data[0].maxminute := 45, [2093].log_data[0].valid := 1, [2093].log_data[1].valid := 1, [2093].log_data[2].valid := 1, [2093].log_data[3].valid := 1, [2093].log_data[4].valid := 1, [2093].log_data[5].valid := 1, [2093].log_data[6].valid := 1, [2093].log_data[7].valid := 1, [2093].log_data[8].valid := 1, [2093].log_data[9].valid := 1, [2093].log_data[10].valid := 1, [2093].log_data[11].valid := 1, [2093].log_data[12].valid := 1, [2093].log_data[13].valid := 1, [2093].log_data[14].valid := 1, [2093].log_data[15].valid := 1, [2093].log_data[16].valid := 1, [2093].log_data[17].valid := 1, [2093].log_data[18].valid := 1, [2093].log_data[19].valid := 1, [2093].time.Year := 2023, [2093].time.Month := 1, [2093].time.Day := 16, [2093].time.Hour := 22, [2093].time.Minute := 49, [2093].time.Second := 59, [2094].log_data[0].min := 1.0, [2094].log_data[0].max := 1.0, [2094].log_data[0].total := 300.0, [2094].log_data[0].time := 300.0, [2094].log_data[0].minminute := 50, [2094].log_data[0].maxminute := 50, [2094].log_data[0].valid := 1, [2094].log_data[1].valid := 1, [2094].log_data[2].valid := 1, [2094].log_data[3].valid := 1, [2094].log_data[4].valid := 1, [2094].log_data[5].valid := 1, [2094].log_data[6].valid := 1, [2094].log_data[7].valid := 1, [2094].log_data[8].valid := 1, [2094].log_data[9].valid := 1, [2094].log_data[10].valid := 1, [2094].log_data[11].valid := 1, [2094].log_data[12].valid := 1, [2094].log_data[13].valid := 1, [2094].log_data[14].valid := 1, [2094].log_data[15].valid := 1, [2094].log_data[16].valid := 1, [2094].log_data[17].valid := 1, [2094].log_data[18].valid := 1, [2094].log_data[19].valid := 1,
        [2094].time.Year := 2023, [2094].time.Month := 1, [2094].time.Day := 16, [2094].time.Hour := 22, [2094].time.Minute := 54, [2094].time.Second := 59, [2095].log_data[0].min := 1.0, [2095].log_data[0].max := 1.0, [2095].log_data[0].total := 300.0, [2095].log_data[0].time := 300.0, [2095].log_data[0].minminute := 55, [2095].log_data[0].maxminute := 55, [2095].log_data[0].valid := 1, [2095].log_data[1].valid := 1, [2095].log_data[2].valid := 1, [2095].log_data[3].valid := 1, [2095].log_data[4].valid := 1, [2095].log_data[5].valid := 1, [2095].log_data[6].valid := 1, [2095].log_data[7].valid := 1, [2095].log_data[8].valid := 1, [2095].log_data[9].valid := 1, [2095].log_data[10].valid := 1, [2095].log_data[11].valid := 1, [2095].log_data[12].valid := 1, [2095].log_data[13].valid := 1, [2095].log_data[14].valid := 1, [2095].log_data[15].valid := 1, [2095].log_data[16].valid := 1, [2095].log_data[17].valid := 1, [2095].log_data[18].valid := 1, [2095].log_data[19].valid := 1, [2095].time.Year := 2023, [2095].time.Month := 1, [2095].time.Day := 16, [2095].time.Hour := 22, [2095].time.Minute := 59, [2095].time.Second := 59, [2096].log_data[0].min := 1.0, [2096].log_data[0].max := 1.0, [2096].log_data[0].total := 300.0, [2096].log_data[0].time := 300.0, [2096].log_data[0].valid := 1, [2096].log_data[1].valid := 1, [2096].log_data[2].valid := 1, [2096].log_data[3].valid := 1, [2096].log_data[4].valid := 1, [2096].log_data[5].valid := 1, [2096].log_data[6].valid := 1, [2096].log_data[7].valid := 1, [2096].log_data[8].valid := 1, [2096].log_data[9].valid := 1, [2096].log_data[10].valid := 1, [2096].log_data[11].valid := 1, [2096].log_data[12].valid := 1, [2096].log_data[13].valid := 1, [2096].log_data[14].valid := 1, [2096].log_data[15].valid := 1, [2096].log_data[16].valid := 1, [2096].log_data[17].valid := 1,
        [2096].log_data[18].valid := 1, [2096].log_data[19].valid := 1, [2096].time.Year := 2023, [2096].time.Month := 1, [2096].time.Day := 16, [2096].time.Hour := 23, [2096].time.Minute := 4, [2096].time.Second := 59, [2097].log_data[0].min := 1.0, [2097].log_data[0].max := 1.0, [2097].log_data[0].total := 300.0, [2097].log_data[0].time := 300.0, [2097].log_data[0].minminute := 5, [2097].log_data[0].maxminute := 5, [2097].log_data[0].valid := 1, [2097].log_data[1].valid := 1, [2097].log_data[2].valid := 1, [2097].log_data[3].valid := 1, [2097].log_data[4].valid := 1, [2097].log_data[5].valid := 1, [2097].log_data[6].valid := 1, [2097].log_data[7].valid := 1, [2097].log_data[8].valid := 1, [2097].log_data[9].valid := 1, [2097].log_data[10].valid := 1, [2097].log_data[11].valid := 1, [2097].log_data[12].valid := 1, [2097].log_data[13].valid := 1, [2097].log_data[14].valid := 1, [2097].log_data[15].valid := 1, [2097].log_data[16].valid := 1, [2097].log_data[17].valid := 1, [2097].log_data[18].valid := 1, [2097].log_data[19].valid := 1, [2097].time.Year := 2023, [2097].time.Month := 1, [2097].time.Day := 16, [2097].time.Hour := 23, [2097].time.Minute := 9, [2097].time.Second := 59, [2098].log_data[0].min := 1.0, [2098].log_data[0].max := 1.0, [2098].log_data[0].total := 300.0, [2098].log_data[0].time := 300.0, [2098].log_data[0].minminute := 10, [2098].log_data[0].maxminute := 10, [2098].log_data[0].valid := 1, [2098].log_data[1].valid := 1, [2098].log_data[2].valid := 1, [2098].log_data[3].valid := 1, [2098].log_data[4].valid := 1, [2098].log_data[5].valid := 1, [2098].log_data[6].valid := 1, [2098].log_data[7].valid := 1, [2098].log_data[8].valid := 1, [2098].log_data[9].valid := 1, [2098].log_data[10].valid := 1, [2098].log_data[11].valid := 1, [2098].log_data[12].valid := 1, [2098].log_data[13].valid := 1,
        [2098].log_data[14].valid := 1, [2098].log_data[15].valid := 1, [2098].log_data[16].valid := 1, [2098].log_data[17].valid := 1, [2098].log_data[18].valid := 1, [2098].log_data[19].valid := 1, [2098].time.Year := 2023, [2098].time.Month := 1, [2098].time.Day := 16, [2098].time.Hour := 23, [2098].time.Minute := 14, [2098].time.Second := 59, [2099].log_data[0].min := 1.0, [2099].log_data[0].max := 1.0, [2099].log_data[0].total := 300.0, [2099].log_data[0].time := 300.0, [2099].log_data[0].minminute := 15, [2099].log_data[0].maxminute := 15, [2099].log_data[0].valid := 1, [2099].log_data[1].valid := 1, [2099].log_data[2].valid := 1, [2099].log_data[3].valid := 1, [2099].log_data[4].valid := 1, [2099].log_data[5].valid := 1, [2099].log_data[6].valid := 1, [2099].log_data[7].valid := 1, [2099].log_data[8].valid := 1, [2099].log_data[9].valid := 1, [2099].log_data[10].valid := 1, [2099].log_data[11].valid := 1, [2099].log_data[12].valid := 1, [2099].log_data[13].valid := 1, [2099].log_data[14].valid := 1, [2099].log_data[15].valid := 1, [2099].log_data[16].valid := 1, [2099].log_data[17].valid := 1, [2099].log_data[18].valid := 1, [2099].log_data[19].valid := 1, [2099].time.Year := 2023, [2099].time.Month := 1, [2099].time.Day := 16, [2099].time.Hour := 23, [2099].time.Minute := 19, [2099].time.Second := 59, [2100].log_data[0].min := 1.0, [2100].log_data[0].max := 1.0, [2100].log_data[0].total := 300.0, [2100].log_data[0].time := 300.0, [2100].log_data[0].minminute := 20, [2100].log_data[0].maxminute := 20, [2100].log_data[0].valid := 1, [2100].log_data[1].valid := 1, [2100].log_data[2].valid := 1, [2100].log_data[3].valid := 1, [2100].log_data[4].valid := 1, [2100].log_data[5].valid := 1, [2100].log_data[6].valid := 1, [2100].log_data[7].valid := 1, [2100].log_data[8].valid := 1, [2100].log_data[9].valid := 1,
        [2100].log_data[10].valid := 1, [2100].log_data[11].valid := 1, [2100].log_data[12].valid := 1, [2100].log_data[13].valid := 1, [2100].log_data[14].valid := 1, [2100].log_data[15].valid := 1, [2100].log_data[16].valid := 1, [2100].log_data[17].valid := 1, [2100].log_data[18].valid := 1, [2100].log_data[19].valid := 1, [2100].time.Year := 2023, [2100].time.Month := 1, [2100].time.Day := 16, [2100].time.Hour := 23, [2100].time.Minute := 24, [2100].time.Second := 59, [2101].log_data[0].min := 1.0, [2101].log_data[0].max := 1.0, [2101].log_data[0].total := 300.0, [2101].log_data[0].time := 300.0, [2101].log_data[0].minminute := 25, [2101].log_data[0].maxminute := 25, [2101].log_data[0].valid := 1, [2101].log_data[1].valid := 1, [2101].log_data[2].valid := 1, [2101].log_data[3].valid := 1, [2101].log_data[4].valid := 1, [2101].log_data[5].valid := 1, [2101].log_data[6].valid := 1, [2101].log_data[7].valid := 1, [2101].log_data[8].valid := 1, [2101].log_data[9].valid := 1, [2101].log_data[10].valid := 1, [2101].log_data[11].valid := 1, [2101].log_data[12].valid := 1, [2101].log_data[13].valid := 1, [2101].log_data[14].valid := 1, [2101].log_data[15].valid := 1, [2101].log_data[16].valid := 1, [2101].log_data[17].valid := 1, [2101].log_data[18].valid := 1, [2101].log_data[19].valid := 1, [2101].time.Year := 2023, [2101].time.Month := 1, [2101].time.Day := 16, [2101].time.Hour := 23, [2101].time.Minute := 29, [2101].time.Second := 59, [2102].log_data[0].min := 1.0, [2102].log_data[0].max := 1.0, [2102].log_data[0].total := 300.0, [2102].log_data[0].time := 300.0, [2102].log_data[0].minminute := 30, [2102].log_data[0].maxminute := 30, [2102].log_data[0].valid := 1, [2102].log_data[1].valid := 1, [2102].log_data[2].valid := 1, [2102].log_data[3].valid := 1, [2102].log_data[4].valid := 1, [2102].log_data[5].valid := 1,
        [2102].log_data[6].valid := 1, [2102].log_data[7].valid := 1, [2102].log_data[8].valid := 1, [2102].log_data[9].valid := 1, [2102].log_data[10].valid := 1, [2102].log_data[11].valid := 1, [2102].log_data[12].valid := 1, [2102].log_data[13].valid := 1, [2102].log_data[14].valid := 1, [2102].log_data[15].valid := 1, [2102].log_data[16].valid := 1, [2102].log_data[17].valid := 1, [2102].log_data[18].valid := 1, [2102].log_data[19].valid := 1, [2102].time.Year := 2023, [2102].time.Month := 1, [2102].time.Day := 16, [2102].time.Hour := 23, [2102].time.Minute := 34, [2102].time.Second := 59, [2103].log_data[0].min := 1.0, [2103].log_data[0].max := 1.0, [2103].log_data[0].total := 300.0, [2103].log_data[0].time := 300.0, [2103].log_data[0].minminute := 35, [2103].log_data[0].maxminute := 35, [2103].log_data[0].valid := 1, [2103].log_data[1].valid := 1, [2103].log_data[2].valid := 1, [2103].log_data[3].valid := 1, [2103].log_data[4].valid := 1, [2103].log_data[5].valid := 1, [2103].log_data[6].valid := 1, [2103].log_data[7].valid := 1, [2103].log_data[8].valid := 1, [2103].log_data[9].valid := 1, [2103].log_data[10].valid := 1, [2103].log_data[11].valid := 1, [2103].log_data[12].valid := 1, [2103].log_data[13].valid := 1, [2103].log_data[14].valid := 1, [2103].log_data[15].valid := 1, [2103].log_data[16].valid := 1, [2103].log_data[17].valid := 1, [2103].log_data[18].valid := 1, [2103].log_data[19].valid := 1, [2103].time.Year := 2023, [2103].time.Month := 1, [2103].time.Day := 16, [2103].time.Hour := 23, [2103].time.Minute := 39, [2103].time.Second := 59, [2104].log_data[0].min := 1.0, [2104].log_data[0].max := 1.0, [2104].log_data[0].total := 300.0, [2104].log_data[0].time := 300.0, [2104].log_data[0].minminute := 40, [2104].log_data[0].maxminute := 40, [2104].log_data[0].valid := 1, [2104].log_data[1].valid := 1,
        [2104].log_data[2].valid := 1, [2104].log_data[3].valid := 1, [2104].log_data[4].valid := 1, [2104].log_data[5].valid := 1, [2104].log_data[6].valid := 1, [2104].log_data[7].valid := 1, [2104].log_data[8].valid := 1, [2104].log_data[9].valid := 1, [2104].log_data[10].valid := 1, [2104].log_data[11].valid := 1, [2104].log_data[12].valid := 1, [2104].log_data[13].valid := 1, [2104].log_data[14].valid := 1, [2104].log_data[15].valid := 1, [2104].log_data[16].valid := 1, [2104].log_data[17].valid := 1, [2104].log_data[18].valid := 1, [2104].log_data[19].valid := 1, [2104].time.Year := 2023, [2104].time.Month := 1, [2104].time.Day := 16, [2104].time.Hour := 23, [2104].time.Minute := 44, [2104].time.Second := 59, [2105].log_data[0].min := 1.0, [2105].log_data[0].max := 1.0, [2105].log_data[0].total := 300.0, [2105].log_data[0].time := 300.0, [2105].log_data[0].minminute := 45, [2105].log_data[0].maxminute := 45, [2105].log_data[0].valid := 1, [2105].log_data[1].valid := 1, [2105].log_data[2].valid := 1, [2105].log_data[3].valid := 1, [2105].log_data[4].valid := 1, [2105].log_data[5].valid := 1, [2105].log_data[6].valid := 1, [2105].log_data[7].valid := 1, [2105].log_data[8].valid := 1, [2105].log_data[9].valid := 1, [2105].log_data[10].valid := 1, [2105].log_data[11].valid := 1, [2105].log_data[12].valid := 1, [2105].log_data[13].valid := 1, [2105].log_data[14].valid := 1, [2105].log_data[15].valid := 1, [2105].log_data[16].valid := 1, [2105].log_data[17].valid := 1, [2105].log_data[18].valid := 1, [2105].log_data[19].valid := 1, [2105].time.Year := 2023, [2105].time.Month := 1, [2105].time.Day := 16, [2105].time.Hour := 23, [2105].time.Minute := 49, [2105].time.Second := 59, [2106].log_data[0].min := 1.0, [2106].log_data[0].max := 1.0, [2106].log_data[0].total := 300.0, [2106].log_data[0].time := 300.0,
        [2106].log_data[0].minminute := 50, [2106].log_data[0].maxminute := 50, [2106].log_data[0].valid := 1, [2106].log_data[1].valid := 1, [2106].log_data[2].valid := 1, [2106].log_data[3].valid := 1, [2106].log_data[4].valid := 1, [2106].log_data[5].valid := 1, [2106].log_data[6].valid := 1, [2106].log_data[7].valid := 1, [2106].log_data[8].valid := 1, [2106].log_data[9].valid := 1, [2106].log_data[10].valid := 1, [2106].log_data[11].valid := 1, [2106].log_data[12].valid := 1, [2106].log_data[13].valid := 1, [2106].log_data[14].valid := 1, [2106].log_data[15].valid := 1, [2106].log_data[16].valid := 1, [2106].log_data[17].valid := 1, [2106].log_data[18].valid := 1, [2106].log_data[19].valid := 1, [2106].time.Year := 2023, [2106].time.Month := 1, [2106].time.Day := 16, [2106].time.Hour := 23, [2106].time.Minute := 54, [2106].time.Second := 59, [2107].log_data[0].min := 1.0, [2107].log_data[0].max := 1.0, [2107].log_data[0].total := 300.0, [2107].log_data[0].time := 300.0, [2107].log_data[0].minminute := 55, [2107].log_data[0].maxminute := 55, [2107].log_data[0].valid := 1, [2107].log_data[1].valid := 1, [2107].log_data[2].valid := 1, [2107].log_data[3].valid := 1, [2107].log_data[4].valid := 1, [2107].log_data[5].valid := 1, [2107].log_data[6].valid := 1, [2107].log_data[7].valid := 1, [2107].log_data[8].valid := 1, [2107].log_data[9].valid := 1, [2107].log_data[10].valid := 1, [2107].log_data[11].valid := 1, [2107].log_data[12].valid := 1, [2107].log_data[13].valid := 1, [2107].log_data[14].valid := 1, [2107].log_data[15].valid := 1, [2107].log_data[16].valid := 1, [2107].log_data[17].valid := 1, [2107].log_data[18].valid := 1, [2107].log_data[19].valid := 1, [2107].time.Year := 2023, [2107].time.Month := 1, [2107].time.Day := 16, [2107].time.Hour := 23, [2107].time.Minute := 59, [2107].time.Second := 59,
        [2108].log_data[0].min := 1.0, [2108].log_data[0].max := 1.0, [2108].log_data[0].total := 300.0, [2108].log_data[0].time := 300.0, [2108].log_data[0].valid := 1, [2108].log_data[1].valid := 1, [2108].log_data[2].valid := 1, [2108].log_data[3].valid := 1, [2108].log_data[4].valid := 1, [2108].log_data[5].valid := 1, [2108].log_data[6].valid := 1, [2108].log_data[7].valid := 1, [2108].log_data[8].valid := 1, [2108].log_data[9].valid := 1, [2108].log_data[10].valid := 1, [2108].log_data[11].valid := 1, [2108].log_data[12].valid := 1, [2108].log_data[13].valid := 1, [2108].log_data[14].valid := 1, [2108].log_data[15].valid := 1, [2108].log_data[16].valid := 1, [2108].log_data[17].valid := 1, [2108].log_data[18].valid := 1, [2108].log_data[19].valid := 1, [2108].time.Year := 2023, [2108].time.Month := 1, [2108].time.Day := 17, [2108].time.Minute := 4, [2108].time.Second := 59, [2109].log_data[0].min := 1.0, [2109].log_data[0].max := 1.0, [2109].log_data[0].total := 300.0, [2109].log_data[0].time := 300.0, [2109].log_data[0].minminute := 5, [2109].log_data[0].maxminute := 5, [2109].log_data[0].valid := 1, [2109].log_data[1].valid := 1, [2109].log_data[2].valid := 1, [2109].log_data[3].valid := 1, [2109].log_data[4].valid := 1, [2109].log_data[5].valid := 1, [2109].log_data[6].valid := 1, [2109].log_data[7].valid := 1, [2109].log_data[8].valid := 1, [2109].log_data[9].valid := 1, [2109].log_data[10].valid := 1, [2109].log_data[11].valid := 1, [2109].log_data[12].valid := 1, [2109].log_data[13].valid := 1, [2109].log_data[14].valid := 1, [2109].log_data[15].valid := 1, [2109].log_data[16].valid := 1, [2109].log_data[17].valid := 1, [2109].log_data[18].valid := 1, [2109].log_data[19].valid := 1, [2109].time.Year := 2023, [2109].time.Month := 1, [2109].time.Day := 17, [2109].time.Minute := 9, [2109].time.Second := 59,
        [2110].log_data[0].min := 1.0, [2110].log_data[0].max := 1.0, [2110].log_data[0].total := 300.0, [2110].log_data[0].time := 300.0, [2110].log_data[0].minminute := 10, [2110].log_data[0].maxminute := 10, [2110].log_data[0].valid := 1, [2110].log_data[1].valid := 1, [2110].log_data[2].valid := 1, [2110].log_data[3].valid := 1, [2110].log_data[4].valid := 1, [2110].log_data[5].valid := 1, [2110].log_data[6].valid := 1, [2110].log_data[7].valid := 1, [2110].log_data[8].valid := 1, [2110].log_data[9].valid := 1, [2110].log_data[10].valid := 1, [2110].log_data[11].valid := 1, [2110].log_data[12].valid := 1, [2110].log_data[13].valid := 1, [2110].log_data[14].valid := 1, [2110].log_data[15].valid := 1, [2110].log_data[16].valid := 1, [2110].log_data[17].valid := 1, [2110].log_data[18].valid := 1, [2110].log_data[19].valid := 1, [2110].time.Year := 2023, [2110].time.Month := 1, [2110].time.Day := 17, [2110].time.Minute := 14, [2110].time.Second := 59, [2111].log_data[0].min := 1.0, [2111].log_data[0].max := 1.0, [2111].log_data[0].total := 300.0, [2111].log_data[0].time := 300.0, [2111].log_data[0].minminute := 15, [2111].log_data[0].maxminute := 15, [2111].log_data[0].valid := 1, [2111].log_data[1].valid := 1, [2111].log_data[2].valid := 1, [2111].log_data[3].valid := 1, [2111].log_data[4].valid := 1, [2111].log_data[5].valid := 1, [2111].log_data[6].valid := 1, [2111].log_data[7].valid := 1, [2111].log_data[8].valid := 1, [2111].log_data[9].valid := 1, [2111].log_data[10].valid := 1, [2111].log_data[11].valid := 1, [2111].log_data[12].valid := 1, [2111].log_data[13].valid := 1, [2111].log_data[14].valid := 1, [2111].log_data[15].valid := 1, [2111].log_data[16].valid := 1, [2111].log_data[17].valid := 1, [2111].log_data[18].valid := 1, [2111].log_data[19].valid := 1, [2111].time.Year := 2023, [2111].time.Month := 1, [2111].time.Day := 17,
        [2111].time.Minute := 19, [2111].time.Second := 59, [2112].log_data[0].min := 1.0, [2112].log_data[0].max := 1.0, [2112].log_data[0].total := 300.0, [2112].log_data[0].time := 300.0, [2112].log_data[0].minminute := 20, [2112].log_data[0].maxminute := 20, [2112].log_data[0].valid := 1, [2112].log_data[1].valid := 1, [2112].log_data[2].valid := 1, [2112].log_data[3].valid := 1, [2112].log_data[4].valid := 1, [2112].log_data[5].valid := 1, [2112].log_data[6].valid := 1, [2112].log_data[7].valid := 1, [2112].log_data[8].valid := 1, [2112].log_data[9].valid := 1, [2112].log_data[10].valid := 1, [2112].log_data[11].valid := 1, [2112].log_data[12].valid := 1, [2112].log_data[13].valid := 1, [2112].log_data[14].valid := 1, [2112].log_data[15].valid := 1, [2112].log_data[16].valid := 1, [2112].log_data[17].valid := 1, [2112].log_data[18].valid := 1, [2112].log_data[19].valid := 1, [2112].time.Year := 2023, [2112].time.Month := 1, [2112].time.Day := 17, [2112].time.Minute := 24, [2112].time.Second := 59, [2113].log_data[0].min := 1.0, [2113].log_data[0].max := 1.0, [2113].log_data[0].total := 300.0, [2113].log_data[0].time := 300.0, [2113].log_data[0].minminute := 25, [2113].log_data[0].maxminute := 25, [2113].log_data[0].valid := 1, [2113].log_data[1].valid := 1, [2113].log_data[2].valid := 1, [2113].log_data[3].valid := 1, [2113].log_data[4].valid := 1, [2113].log_data[5].valid := 1, [2113].log_data[6].valid := 1, [2113].log_data[7].valid := 1, [2113].log_data[8].valid := 1, [2113].log_data[9].valid := 1, [2113].log_data[10].valid := 1, [2113].log_data[11].valid := 1, [2113].log_data[12].valid := 1, [2113].log_data[13].valid := 1, [2113].log_data[14].valid := 1, [2113].log_data[15].valid := 1, [2113].log_data[16].valid := 1, [2113].log_data[17].valid := 1, [2113].log_data[18].valid := 1, [2113].log_data[19].valid := 1, [2113].time.Year := 2023,
        [2113].time.Month := 1, [2113].time.Day := 17, [2113].time.Minute := 29, [2113].time.Second := 59, [2114].log_data[0].min := 1.0, [2114].log_data[0].max := 1.0, [2114].log_data[0].total := 300.0, [2114].log_data[0].time := 300.0, [2114].log_data[0].minminute := 30, [2114].log_data[0].maxminute := 30, [2114].log_data[0].valid := 1, [2114].log_data[1].valid := 1, [2114].log_data[2].valid := 1, [2114].log_data[3].valid := 1, [2114].log_data[4].valid := 1, [2114].log_data[5].valid := 1, [2114].log_data[6].valid := 1, [2114].log_data[7].valid := 1, [2114].log_data[8].valid := 1, [2114].log_data[9].valid := 1, [2114].log_data[10].valid := 1, [2114].log_data[11].valid := 1, [2114].log_data[12].valid := 1, [2114].log_data[13].valid := 1, [2114].log_data[14].valid := 1, [2114].log_data[15].valid := 1, [2114].log_data[16].valid := 1, [2114].log_data[17].valid := 1, [2114].log_data[18].valid := 1, [2114].log_data[19].valid := 1, [2114].time.Year := 2023, [2114].time.Month := 1, [2114].time.Day := 17, [2114].time.Minute := 34, [2114].time.Second := 59, [2115].log_data[0].min := 1.0, [2115].log_data[0].max := 1.0, [2115].log_data[0].total := 300.0, [2115].log_data[0].time := 300.0, [2115].log_data[0].minminute := 35, [2115].log_data[0].maxminute := 35, [2115].log_data[0].valid := 1, [2115].log_data[1].valid := 1, [2115].log_data[2].valid := 1, [2115].log_data[3].valid := 1, [2115].log_data[4].valid := 1, [2115].log_data[5].valid := 1, [2115].log_data[6].valid := 1, [2115].log_data[7].valid := 1, [2115].log_data[8].valid := 1, [2115].log_data[9].valid := 1, [2115].log_data[10].valid := 1, [2115].log_data[11].valid := 1, [2115].log_data[12].valid := 1, [2115].log_data[13].valid := 1, [2115].log_data[14].valid := 1, [2115].log_data[15].valid := 1, [2115].log_data[16].valid := 1, [2115].log_data[17].valid := 1, [2115].log_data[18].valid := 1,
